(* IEC 61131-3 sources: ml2plc/benchmarks/st (part 24) *)

    bias_8 : ARRAY[0..63] OF REAL := [-0.00346507085, 0.0794098824, -0.0815823004, -0.0197601747, -0.0118380254, 0.0312293377, -0.00609452976, 0.00358696282, 0.00419461308, -0.0723088458, 0.0482314527, 0.0938620642, -0.0692073926, 0.0194631442, -0.0589119196, 0.0299020465, -0.00631620362, 0.00955793448, -0.0159860123, 0, -0.00618809368, 0.0138237355, 0.00124220713, -0.0202849712, -0.00431400631, -0.0275725052, 0.111446135, 0.11047177, 0, 0.0995986015, 0.0175163615, 0.0613925792, -0.00830586068, 0.00282396353, -0.0744342729, -0.0211106688, 0.0866850466, 0.0997213498, -0.00675268006, -0.0535650924, -0.0118874479, -0.0482638218, 0.00823871326, 0.0484990887, -0.0278981514, 0.0414009988, 0.0608626865, 0.0968099013, -0.0129826535, -0.0369008854, 0.00364142703, -0.0370340049, -0.00600347202, -0.0126274861, 0.0921183825, -0.0980235487, 0.00168389722, 0.0823842064, 0.0339883827, 0.0445966795, 0.0921582058, -0.0254019089, -0.0172969531, 0.0778813958];

    weights_11 : ARRAY[0..4095] OF REAL := [0.152399674, -0.263345957, -0.224488631, -0.188193366, -0.0617991723, 0.148717895, 0.0324863903, 0.114666007, -0.289823532, 0.0125278663, -0.0137963807, -0.022444414, 0.110561207, 0.119829476, 0.334477097, -0.139504924, -0.0269849207, 0.113053806, -0.0107069612, -0.180623204, 0.0457108654, -0.214532733, 0.0401020236, 0.00631321967, -0.167630613, -0.0481288582, 0.195484549, 0.111929268, -0.0581923984, 0.0258115064, 0.238763675, 0.0641915128, -0.0806587264, -0.224124625, -0.0460969172, 0.091414094, -0.013553381, -0.043530602, -0.0263040792, 0.140525028, -0.0622836426, 0.15601474, -0.497485936, 0.129424945, -0.170885473, -0.125799641, -0.339268953, 0.0710499883, -0.116152979, -0.0266817547, 0.126233891, 0.131714255, 0.290685475, 0.165184066, 0.283396602, -0.059989959, 0.0141595677, -0.136663362, 0.20351474, 0.0463219136, 0.00223265006, 0.0316324756, 0.182196692, 0.341547728, 0.0614045113, -0.00371772563, -0.275792897, -0.193623677, -0.0266438629, -0.103982933, 0.0405711122, -0.00346332369, 0.0464573167, 0.000740021234, -0.303002685, 0.0795986727, -0.0327266343, 0.0721366256, 0.147136018, -0.105440497, 0.101954572, 0.0728471428, -0.0363206528, -0.0158560108, -0.330246508, -0.212550044, -0.093112044, -0.197731018, -0.125574902, -0.078097105, 0.034774553, -0.262974173, 0.15699707, 0.14151752, -0.0313425213, -0.0470193997, 0.19462584, -0.255247116, 0.357496887, 0.000614301243, -0.195358515, 0.0303748176, -0.175757021, -0.0335321315, -0.0249454323, 0.0811241418, 0.0762640387, 0.116933405, -0.128208607, 0.00518320873, -0.029634852, 0.11359746, 0.017268436, -0.104347244, -0.115615718, 0.202678129, 0.10678266, 0.0986468866, 0.190590888, 0.0687514096, 0.0356852412, -0.0412406325, 0.0757317245, 0.0352434814, -0.342369705, -0.0480474308, 0.266226262, 0.0569148995, 0.0286941677, -0.2472938, 0.0204578005, 0.0296292026, -0.0654909462, -0.10515099, 0.151057318, -0.0363138504, 0.00139550562, 0.0611258186, 0.0148243103, 0.227309123, -0.0798782185, -0.11899174, -0.157541484, 0.314520597, 0.170248464, 0.265226632, 0.0593360811, -0.0398373678, 0.0081351446, -0.0901603773, 0.18755962, 0.00631602108, -0.207302138, 0.103253566, -0.240270436, -0.0895837396, -0.105462186, -0.135611624, -0.0793325603, -0.0249736756, -0.13815324, -0.0941773206, -0.189351335, -0.112737559, 0.293767184, 0.0163262729, -0.175204575, -0.0996527299, 0.231760427, -0.0418962091, -0.0648548007, 0.268336385, -0.032381732, 0.245270595, 0.0585076436, -0.0289969705, 0.232107788, 0.279983878, -0.011282769, -0.121292524, -0.295017779, -0.131171674, 0.0821883231, 0.216307148, -0.0106242169, 0.00658608973, -0.21936737, -0.139937028, 0.182932571, 0.233257622, -0.286341697, 0.246410012, -0.0386230387, 0.0858042613, -0.0830237195, -0.110467531, 0.0558926836, -0.0293775387, -0.216672435, 0.134263664, -0.0869384855, -0.0198220555, -0.0998319387, 0.122479506, 0.124716364, 0.12669073, -0.165978372, -0.0657829642, 0.0525778681, 0.0783382952, 0.0370095335, 0.141239166, 0.0418702848, 0.0749414936, 0.240086794, 0.0674306303, 0.0347193331, -0.0469557568, 0.041893255, 0.090664953, 0.0798208192, -0.124962248, -0.0150589822, 0.0606806017, -0.212737143, 0.0127978772, -0.0479948185, 0.193862215, 0.18940939, 0.110280916, 0.00163242826, -0.0205761306, -0.129006281, -0.141371146, 0.147304669, 0.0262788441, 0.167370602, -0.141203105, 0.200771987, -0.234238222, -0.149722278, 0.23931098, 0.0104937805, -0.266669959, -0.164157122, -0.041039072, -0.250695556, -0.112417288, 0.193107903, 0.140542001, 0.0903390646, -0.230039254, 0.0777369738, 0.260997742, 0.0930059701, 0.138459459, 0.0424353629, 0.171048418, 0.156789139, 0.0312985368, 0.133111879, -0.120839193, 0.0985307842, -0.175964057, 0.122762412, -0.117720641, -0.129174918, -0.104449466, -0.144933715, -0.215081707, 0.0680070445, -0.129005954, 0.0603452325, -0.0575148351, -0.203575164, -0.0453374311, 0.155170351, 0.106897905, 0.0749150291, -0.144247919, -0.171046615, -0.132302389, -0.147862911, 0.00684731873, -0.0410480648, 0.15876098, -0.190579101, 0.0498549677, 0.0963715315, 0.086084798, -0.0875354186, -0.153710201, 0.145764962, 0.0200527348, -0.100025706, -0.135493338, -0.0464859232, 0.00132688298, -0.0185684748, 0.0582565144, 0.187669724, -0.0816467628, -0.0872224793, 0.157934099, 0.0402881019, -0.0318563916, -0.142950997, -0.11230398, -0.0497585908, 0.161313683, -0.1942278, -0.0826544166, -0.0122894971, 0.0872979611, 0.0720221922, 0.0849900693, -0.177533969, -0.152409315, -0.100491337, -0.0112174684, 0.106480442, -0.0379864834, 0.0722993612, 0.163500831, 0.18924883, -0.135068297, 0.0942396447, 0.0284191072, -0.0632716715, -0.138580009, 0.193715364, -0.150715292, 0.0303814765, 0.111110657, 0.117106274, -0.0263905209, 0.0506038666, 0.0267103072, 0.0400604308, 0.154954746, 0.108434454, 0.0550541244, 0.0168840457, 0.0785695761, 0.0604145676, 0.144188315, -0.206482708, 0.0983125418, -0.0374258012, -0.00447623339, 0.205374479, -0.0380841345, 0.0740306601, -0.0350800455, 0.0866823494, -0.0981449634, 0.0656447932, 0.0974652469, 0.0593180098, -0.0401085094, -0.0922544375, 0.0644713044, -0.0637705103, 0.205211937, 0.27076602, 0.0604185574, 0.245794445, -0.0236300994, -0.027567558, 0.1355685, 0.0849664137, -0.138995841, 0.159796208, 0.0539290234, -0.0213833489, 0.0917554945, -0.193392858, 0.0205196254, -0.154481247, -0.0105813192, 0.158501342, 0.01522783, -0.0629718155, -0.222794086, -0.138768524, 0.00203081919, 0.170994595, -0.0148755405, 0.0800000504, 0.194157824, -0.113540575, 0.0917406157, 0.238140926, 0.00717910752, 0.21342735, 0.0675954148, -0.0781002492, 0.179200038, -0.0140909683, 0.217517018, -0.0182730798, 0.154534876, 0.130978897, -0.15910472, -0.242845848, 0.192364007, -0.0712619573, -0.172466293, 0.153321937, 0.196527407, -0.14488329, 0.0236006379, 0.0861952752, -0.0437985249, 0.175121501, -0.0954023749, -0.114573762, 0.143516839, 0.00525142904, 0.126135498, -0.116257451, 0.109212697, 0.0145286033, 0.104307882, -0.0975407884, -0.164253727, 0.0486553423, 0.0687329695, 0.187514946, -0.049572818, 0.0788708553, -0.0701822415, -0.045390375, 0.100607939, -0.0249090847, 0.0791288838, 0.154155806, 0.232392356, 0.110889055, 0.0298407078, -0.0190417878, -0.0341505446, -0.22469382, 0.0715206563, -0.109233215, 0.0421755537, 0.0418922678, -0.0328179933, -0.161357954, 0.0284879543, 0.0438218452, 0.257945627, 0.227448493, -0.129958495, -0.392283171, 0.109769329, -0.0173306819, 0.0859658271, 0.108519241, -0.0660175383, -0.0608303361, -0.0360111594, -0.0876427889, 0.190083712, 0.0288716163, 0.238107309, 0.136543661, -0.00705705583, -0.0259979162, -0.00647293031, 0.069024533, 0.0381969362, -0.152234167, 0.295585841, -0.401145488, -0.108133636, 0.209102049, 0.0307547674, 0.147690207, 0.128031835, -0.0473762713, -0.147987187, -0.164643124, -0.059981253, -0.14839074, -0.0456473343, -0.335970312, 0.0270624142, 0.273908377, 0.0461861901, -0.221928775, 0.151594713, 0.0270567555, 0.0552504733, 0.288964689, -0.075935334, 0.270585835, 0.235102609, 0.181183606, -0.116892524, 0.0349841826, -0.0259137452, -0.310423553, -0.0737684369, -0.224190742, 0.102769867, 0.148424283, -0.00051581359, 0.109018147, 0.131758898, -0.241935253, 0.0429472104, -0.192998812, -0.156563684, -0.199549347, -0.0259795301, 0.118114009, -0.202294961, 0.00430562347, -0.0795410797, -0.186826259, -0.12402641, -0.0973436236, 0.062623024, 0.0698438436, -0.0140991006, 0.0761193931, -0.157981157, 0.054249879, -0.0833289996, -0.119116187, -0.175815642, -0.193181172, -0.0350408033, 0.0374635346, -0.148473918, -0.111192934, -0.110237554, 0.0392782576, 0.0543338954, -0.212789983, 0.214189187, 0.261465758, 0.0389742181, -0.0119669382, -0.041862458, 0.0934221447, 0.154760599, 0.104591891, 0.135659441, 0.124115832, 0.125245571, -0.0981265381, -0.173501864, -0.225834534, -0.040620435, -0.0631992593, 0.11226812, -0.151412457, 0.0888080448, 0.130535215, 0.114341483, 0.0704539269, 0.238751054, -0.0625069663, 0.183925942, 0.162767082, -0.0624889433, 0.18303372, 0.0478743874, -0.214895129, 0.150446177, -0.0400604196, 0.164489478, 0.156864062, 0.280662, 0.0744856521, -0.109412298, 0.222006962, -0.188556612, 0.257241905, 0.00763767865, -0.0429345556, 0.000701996032, -0.256307662, -0.0537884794, 0.258199453, -0.145994559, 0.0452899151, 0.0317057781, -0.0876930654, 0.08571475, -0.092731908, 0.184803054, 0.18809928, 0.0703473389, -0.00392604945, 0.142104432, 0.160575241, -0.0699259192, 0.196616039, -0.160764754, -0.202707544, 0.150236309, -0.194807246, -0.142325938, -0.240276873, -0.0591731966, -0.0514629297, 0.00134343619, -0.166902661, -0.188654795, 0.0843883976, 0.0013771971, 0.169252023, -0.161208317, 0.208919898, -0.118219167, -0.24853687, 0.147254348, -0.040950682, -0.104150467, -0.182231963, -0.162871018, 0.0433620438, 0.126293465, -0.166178107, -0.186834484, -0.22719419, -0.216035366, -0.311863422, 0.10080345, -0.10563679, -0.21303615, 0.0257087015, 0.063385427, 0.0836621374, 0.137088358, 0.0247118175, 0.157823056, -0.162809089, 0.274433285, -0.0909785628, 0.219206274, -0.150779128, -0.206102833, 0.0196267851, 0.215949804, -0.080320105, 0.0171771869, -0.126778483, -0.169971392, -0.0758564174, 0.037309479, -0.184586704, -0.176283911, -0.0172518641, -0.223967373, 0.0620737523, -0.210962385, -0.0175580438, -0.198382184, -0.133766785, -0.192560017, 0.00918835402, -0.0767401755, 0.136367351, 0.171674535, 0.183295757, 0.220561728, -0.0821217224, 0.1140071, -0.127449334, -0.151443526, 0.118891813, 0.0171878282, -0.027197564, -0.0242941491, -0.232013106, -0.109213538, -0.117022179, 0.0856248662, -0.151049286, 0.142516539, 0.125007212, -0.156722993, 0.266981691, -0.130809814, -0.0616114177, -0.0442247763, 0.0877789408, 0.0459268093, 0.225089535, 0.059550181, -0.0352692939, -0.0199252516, -0.140248358, -0.181541502, -0.0301125441, 0.114853002, -0.155363366, 0.120270431, -0.119383417, 0.15385288, -0.137697816, 0.0990949422, 0.139819413, 0.101220191, 0.0159896575, -0.0617526323, -0.0679681972, 0.113188118, -0.042417895, 0.0258083455, -0.169725969, 0.075258702, -0.0537487082, -0.149268836, 0.109437704, -0.116023861, 0.0976026133, -0.215568498, -0.257916421, -0.0836541727, 0.0753511712, 0.194070086, 0.0318242721, 0.0160240829, 0.0868645757, -0.188116699, 0.181180835, -0.207172692, 0.110726506, 0.171905503, -0.121312834, 0.00326830451, -0.134259403, -0.244052947, 0.156338409, 0.239065826, 0.0572260544, 0.22199899, 0.0920382291, -0.0747542828, 0.0250579547, -0.209005356, 0.314894259, -0.0127276182, 0.188592002, -0.105892763, -0.203456968, 0.218186542, -0.0714133903, -0.090361774, -0.0645971596, 0.0143091576, 0.298341304, 0.159289271, 0.0570015721, -0.199153751, 0.019798452, -0.0419481322, -0.128920168, 0.0999377146, -0.245023876, -0.0517567694, 0.247462109, -0.070638895, -0.0811767727, -0.128980458, 0.11074882, 0.0168372188, 0.0593690798, 0.175101206, -0.054478053, 0.022643229, -0.307910532, -0.0983424112, 0.0169419218, -0.131076947, 0.295372337, -0.176049858, -0.0388735868, 0.261773378, 0.186196834, 0.0407921039, -0.060955897, 0.0722839534, 0.1541913, 0.118314162, 0.185275882, -0.0770900249, -0.186694846, 0.118786186, -0.022491321, -0.0364597216, 0.089644663, 0.0571428053, -0.253871858, -0.0122213988, 0.204711184, 0.312439799, -0.320880443, -0.27240929, 0.122102626, -0.273709536, -0.0164961014, 0.0607479513, 0.291678041, 0.223591253, -0.198138237, -0.118850462, -0.238560677, 0.323092818, 0.0589599535, -0.194248945, 0.00573190255, -0.0346102566, 0.00809514709, -0.1437345, -0.0768056959, -0.0114840511, 0.14923422, -0.0970238969, -0.0471924804, 0.0891452581, 0.176614508, -0.150917053, 0.31215173, -0.0488434397, 0.0310474988, 0.13556391, -0.210260242, 0.265471876, 0.127534941, 0.00403250754, 0.210733801, 0.0956179649, 0.0654093474, 0.0347067229, 0.0318550393, 0.248021692, 0.0198314767, -0.115047991, 0.108949013, -0.10042078, -0.29889968, 0.0146387629, -0.141234264, 0.204530731, -0.144104674, 0.105720773, -0.23340179, 0.0790494978, 0.18509376, -0.206608996, -0.0394043922, -0.0189410113, -0.230545685, -0.198211581, 0.220677823, -0.0647635758, -0.195251271, 0.201641157, -0.177163646, -0.095896475, 0.0920335501, -0.138604224, -0.109693781, 0.236355498, 0.0536849797, 0.115611076, 0.212027684, 0.0571522713, 0.240873307, -0.0458607674, 0.310614586, 0.233346224, 0.0570905395, 0.130410984, 0.169783399, 0.0727831423, -0.0302463956, -0.30536887, 0.0152019113, 0.163850963, -0.109125808, 0.0144169629, 0.132228628, -0.0707990453, 0.193070427, 0.165563926, 0.0941457525, -0.0627072603, 0.0423249342, -0.111638814, -0.0591745116, -0.0470574982, 0.29292962, 0.0765838027, -0.142371729, -0.112034045, -0.0560461804, 0.156755283, -0.235810399, -0.201336101, -0.125491038, 0.201229259, 0.123228803, -0.238689259, 0.0129049234, 0.0961765721, 0.0151871378, 0.266222477, 0.186487585, -0.217119902, -0.0869368389, 0.124067664, -0.065676488, 0.140951827, -0.198084503, -0.178457528, 0.0855591595, 0.1007246, -0.0287072621, 0.0854200944, -0.178427383, 0.0386579223, -0.0619194172, 0.09910997, -0.129233211, -0.068861261, 0.13413316, 0.139778435, 0.0833287686, 0.0622766875, 0.235616207, 0.201298133, -0.182556123, -0.00869753398, -0.047157418, 0.268308789, -0.225152835, 0.0152922235, 0.153030574, -0.0839851871, 0.167121798, -0.0833399519, 0.093423374, -0.0923105478, 0.178122193, -0.203960165, 0.0267385971, 0.0512525626, -0.22356531, 0.056387879, -0.0550887249, 0.161965206, -0.195818886, -0.0647771284, -0.182523564, 0.17741926, -0.116015404, -0.0489375815, -0.202825278, 0.147160143, 0.191247597, 0.0707065612, -0.00766302971, 0.170157924, 0.0735885873, -0.141567349, -0.21014148, -0.129353657, 0.0956847668, 0.0227197595, 0.0941244364, -0.0791912824, 0.107957929, 0.199303105, 0.0537132025, 0.0155240446, -0.147489786, 0.0846396238, -0.0715232193, 0.182592198, 0.00312403357, 0.0118206823, 0.0933757424, 0.162187204, -0.0768953189, 0.130623519, -0.154309347, -0.0370425209, 0.225373268, -0.0371935703, -0.512049019, 0.0894301012, 0.149142876, 0.0406918228, 0.054195568, -0.222945645, 0.125597313, -0.121843651, -0.192063659, 0.022529887, -0.129418507, 0.100320496, 0.14389959, 0.100439146, 0.211798623, -0.139967546, 0.104904346, -0.0939587057, 0.127366856, 0.138831839, 0.0239571333, -0.00880390406, -0.0611199997, -0.10359811, -0.0635057986, -0.00202414393, 0.188975051, 0.18646647, -0.133227944, 0.0697101131, -0.0743370131, 0.0876726359, 0.174912781, 0.132824585, 0.00545993866, -0.000499482965, 0.169128001, 0.219260916, 0.214551806, -0.0652708858, -0.0217023604, -0.193402603, 0.00403163396, -0.117414609, -0.0933148414, 0.00748919882, 0.200135365, -0.141633987, -0.214732349, -0.091433309, 0.204348087, -0.0532101393, 0.154062733, 0.248481318, -0.13802442, 0.192950904, 0.16888696, 0.149313912, -0.222851619, 0.153076321, 0.182242945, 0.185836926, 0.141479209, -0.0413135886, -0.0169824678, -0.0272292644, 0.089787066, -0.0702687651, 0.158348948, -0.0452950932, -0.0598885454, -0.174950615, 0.291644782, -0.0561419651, 0.0800843909, -0.215036035, 0.13363564, -0.103067927, -0.0768741667, -0.0631346405, 0.0626737475, 0.15906544, -0.327983201, -0.123729207, 0.19425182, -0.14580068, -0.110915102, -0.0493397824, 0.0671491474, 0.00072730938, 0.0883379132, 0.123690397, 0.189004809, 0.0893278271, -0.114139549, 0.308739871, 0.0107161012, 0.118270479, -0.337565839, 0.261260688, -0.0494029, -0.0752659142, 0.238311097, -0.108185798, -0.12475723, -0.0681707337, 0.0807750225, 0.0104115838, -0.0831196159, -0.161203995, 0.0769510195, -0.178012058, 0.165514678, -0.0196140297, -0.0373411514, -0.0155290961, -0.161595047, -0.0622068048, -0.291716814, 0.218920842, -0.128163859, 0.044695992, -0.187777534, -0.105463572, -0.0571242459, -0.0119509697, 0.00533423526, -0.0132009489, 0.161444128, 0.190533608, 0.136306271, 0.158209473, 0.215961605, -0.0804739892, 0.117368713, 0.126664549, 0.133364782, 0.152663857, 0.136497244, -0.336019129, 0.150216475, 0.20953989, -0.0419718549, 0.00763540342, 0.0507058874, 0.0899446309, -0.0746354163, 0.126670465, 0.0997138247, -0.131774053, 0.18959567, 0.186503679, 0.0671444461, 0.107626587, 0.125563666, -0.0331348479, -0.0831428245, -0.0118116708, 0.13317202, 0.179913059, -0.00435783528, -0.103403352, -0.169043481, 0.134726152, -0.143405557, -0.143480599, 0.145388424, 0.0501072556, -0.100935332, 0.0670109838, -0.0547590144, -0.11869137, -0.164782315, 0.14261204, 0.0516628996, -0.0139837861, 0.158076271, -0.0323812068, -0.0253638402, -0.0481653959, -0.166442499, 0.0914008841, -0.126121193, 0.10642685, 0.080969587, 0.195150837, -0.0635801703, 0.0927808583, 0.0660431832, -0.113444202, 0.2108161, 0.0454176217, 0.207712188, -0.158912182, -0.149667591, 0.225732028, -0.144124746, 0.220306486, 0.187320516, -0.056225121, 0.190556765, -0.184439331, -0.128877133, -0.0283655971, 0.148606017, -0.103650376, 0.0173259694, 0.0809403509, 0.00934745371, -0.129418105, -0.0100147277, 0.0515523404, 0.00264053047, -0.133236319, 0.213405624, 0.200618967, 0.011354222, 0.0573964044, 0.0985980853, 0.00135266967, -0.129998296, 0.151727006, 0.204372659, 0.200007543, 0.21404855, 0.189805731, 0.172358885, -0.0890808403, 0.0522677153, 0.107005432, 0.113238558, 0.0461152345, 0.119334862, 0.113662854, -0.202756092, 0.122567102, 0.156569704, 0.0166884214, -0.127153099, 0.130326495, -0.162898168, 0.0981043428, 0.199507132, -0.092357628, -0.0304451138, -0.156488106, 0.0427581519, -0.213457823, 0.157986298, 0.212126359, -0.191093981, -0.0687070787, -0.155501977, 0.075762704, 0.202147499, -0.0100540668, -0.0357479602, -0.165612519, 0.0348113328, 0.0888052136, 0.0522147566, 0.00634533167, -0.000127598643, 0.0748969465, 0.0386748761, 0.0424322337, 0.212277904, -0.0906898081, -0.0402118266, -0.14763388, -0.163068712, -0.00134003162, 0.0113786161, -0.114206046, 0.0614237338, -0.143889531, -0.096885711, 0.20141612, -0.20934172, 0.159835026, 0.0288719237, 0.0186812729, 0.0141171068, 0.202441737, -0.00636282563, -0.0913520604, -0.00343427062, -0.0776682198, 0.114591286, 0.178352684, 0.072447516, 0.207320198, -0.164817482, -0.133918926, 0.0607623905, 0.133606508, 0.108131513, -0.00368179381, -0.0975685716, -0.18251574, -0.12751992, 0.217671528, -0.00256840885, 0.0633859858, 0.0459913127, -0.0114317834, 0.019155506, -0.0564544499, -0.173174202, -0.0360071398, -0.161694646, -0.201523215, 0.143933117, -0.0519516505, -0.189812288, 0.0398772061, -0.0408333391, -0.180227458, 0.141621813, -0.115172304, -0.121136017, -0.0121303732, -0.204050809, -0.0434726924, -0.046715267, -0.0699533895, 0.171459943, -0.144236326, -0.0683937967, -0.0708762109, -0.102386728, -0.0776161775, -0.193716198, 0.186093926, 0.0237003118, 0.121066563, -0.125280246, 0.0977233648, -0.0399483182, -0.0141839087, 0.145612508, 0.0374964625, 0.0779918507, -0.0435630977, 0.0875028968, 0.071565561, -0.0101307984, 0.165002391, 0.201880664, 0.00914894603, 0.186509728, 0.170419008, -0.00774519145, 0.0486198589, -0.257243395, 0.0580342449, -0.123784639, 0.13865912, -0.172557667, 0.151741877, -0.101602815, 0.110366128, -0.120282121, 0.0840358585, -0.13807863, 0.135065734, 0.152518809, -0.213707358, 0.157859072, -0.0512838028, -0.119913951, -0.0603275895, -0.0344250649, 0.0280932616, -0.113776729, 0.00914250128, 0.169182256, -0.0726605803, -0.118695714, -0.162195101, 0.109512694, 0.214561909, 0.201593056, -0.0490923934, 0.231536657, 0.000906694273, -0.0773898289, 0.229626477, 0.292316675, 0.0434411876, 0.0439935587, -0.171945095, 0.168419257, 0.138824657, 0.187337905, -0.121906206, -0.121290758, 0.0895823315, -0.205835402, -0.102580823, -0.064769879, 0.0918552354, -0.0006545863, 0.0484051257, 0.00231042434, -0.1427017, -0.00512752309, -0.118499592, 0.167649359, 0.173335105, 0.0724587515, -0.0639462695, 0.189106256, -0.0253329333, -0.167535514, 0.199837193, 0.054232005, 0.173054591, 0.208212107, 0.063709937, 0.178403363, 0.102365844, -0.145370528, -0.0627328828, 0.204421952, -0.217216507, 0.152429745, 0.177940995, 0.123621874, 0.161663517, -0.0583134182, 0.113821968, 0.147727966, -0.0192146897, 0.120329253, -0.206288442, 0.118907943, 0.0558229275, -0.119626381, 0.115259588, -0.123966016, 0.189842731, 0.304001242, -0.133949921, -0.00190896366, 0.111900635, 0.194404766, 0.129541457, -0.0793663859, 0.0952215493, -0.205361709, 0.0308174528, 0.276944697, 0.150184885, 0.0571603253, -0.0862910375, -0.209261745, -0.00469737314, -0.107266292, -0.0262841173, -0.21763204, 0.0261462647, 0.0255539753, 0.159364834, 0.0638701171, -0.133363664, 0.166979283, -0.191513494, 0.167016715, -0.201660112, 0.0460934602, -0.00581953721, 0.00407372508, -0.078385748, 0.176348567, 0.261097163, 0.0668909401, 0.0932687446, 0.268428653, 0.111295953, -0.0538752489, -0.0353972577, -0.0643084422, 0.0826371983, 0.241673946, 0.0859841257, 0.0413935967, 0.192854241, -0.0863617063, 0.102388531, 0.0939005539, 0.110310666, 0.0338847861, -0.0237080809, 0.192427814, 0.00698334165, 0.0662905425, -0.134980679, -0.00617967499, 0.190878674, -0.00159786642, 0.0727328956, -0.240946233, 0.196102977, -0.0931468382, 0.0836528018, 0.103284612, -0.239004865, 0.0113834683, -0.129806876, 0.14836894, -0.232858315, 0.089459613, -0.179351673, 0.144995049, 0.196424425, -0.0279766843, 0.132153019, -0.105318397, 0.187499374, -0.00858527701, -0.0920507312, -0.11234127, -0.0994759649, 0.175084785, -0.0811289176, -0.100668162, -0.387158185, 0.153878331, -0.178559199, -0.119826905, -0.0257519037, 0.202533126, -0.165797308, 0.1972083, 0.0326090157, 0.191457987, 0.208948106, -0.0303138606, -0.168486714, -0.212763578, -0.00552030979, -0.0189667419, 0.196747944, 0.209965065, -0.14008227, -0.356117338, 0.0720864087, 0.2261962, 0.262177914, 0.190582126, 0.125341758, 0.131352305, -0.0850886703, 0.105056457, 0.0996146277, -0.364396185, -0.1066579, -0.145678446, 0.0647635385, 0.0825714245, -0.0452001728, 0.13121967, -0.145201892, 0.102415368, 0.160855427, -0.1157851, 0.176233247, -0.106195346, -0.17459546, 0.0715932772, 0.0647462085, -0.0499108769, 0.0551721789, 0.0756226256, -0.115369171, 0.115483992, 0.182759956, 0.134363547, 0.19813326, -0.00339539489, 0.22427693, 0.0874575227, -0.0538085252, 0.0250612367, 0.194358304, 0.0420459919, -0.197343454, 0.15234834, -0.0194482468, 0.207918748, -0.370312631, -0.191926241, -0.238808528, -0.0383893885, 0.126615122, -0.0540592968, -0.207585737, -0.0226110499, 0.0861546621, 0.258043557, 0.30580011, -0.265124172, -0.172527641, -0.0776732266, 0.0940554887, -0.0529039092, 0.22364676, -0.0504839607, -0.111994199, 0.0752739981, 0.167051509, 0.231486157, 0.222942859, -0.0696845353, -0.151163772, 0.250781924, -0.146447971, -0.0967529416, 0.184217557, -0.300973266, -0.126572028, 0.215180457, 0.187338904, 0.185731187, -0.11665196, 0.000876162725, -0.0202561766, 0.125354245, 0.10827215, -0.160607785, 0.188338622, 0.0980067775, 0.0324687324, -0.219831422, -0.168211251, 0.200699002, 0.1139713, -0.216335818, -0.0309214499, 0.0763551295, 0.0451243334, 0.0868523866, -0.000636569108, 0.0952483416, -0.11416243, -0.125886872, 0.0755488724, 0.107398666, -0.0849267319, 0.0167402681, -0.368645281, -0.106054433, -0.136857152, -0.113142923, -0.140909985, -0.0106369946, -0.0734956935, -0.242627531, -0.163561374, 0.0919052735, 0.125031963, -0.043657735, 0.0146407625, 0.153221101, 0.0668651685, -0.190944195, 0.0788392946, -0.0817975849, 0.124928646, -0.361474574, 0.110909373, -0.255627602, -0.142462447, 0.0353607163, -0.252555937, 0.194031313, -0.0276524629, -0.0741961077, 0.0262450166, -0.102495871, 0.107768953, 0.141406447, -0.322431296, 0.174083382, -0.174821675, -0.395054817, -0.0608991683, -0.341402888, -0.146280155, -0.290810555, -0.0700072646, 0.0340672284, 0.114190154, 0.212211475, -0.29652983, 0.0295428969, 0.194639176, -0.0198184811, 0.133799478, 0.138498858, -0.182915777, 0.0482293516, 0.0976990163, -0.18222487, 0.0835105181, -0.106537037, -0.0591551289, -0.115260668, -0.11497248, 0.0435057431, -0.159548879, -0.105683692, -0.260151893, 0.0550674088, -0.0321849883, -0.0744472593, 0.00243522367, -0.181820303, 0.252596408, 0.270988226, 0.168165222, 0.0595975779, 0.0989734977, 0.17273213, 0.0179654639, 0.013571118, 0.0022207133, -0.0643146485, 0.14008981, -0.0777452365, 0.134650469, -0.155961126, 0.0555896498, -0.0966854021, 0.0125770848, -0.000214683023, -0.151022673, 0.196903691, -0.115989923, 0.262134969, -0.0680010691, -0.224485368, -0.199625343, -0.210131735, -0.0643070862, 0.0685092211, -0.413198173, 0.0757171661, 0.0919734463, -0.359562606, -0.201385498, 0.0115947183, 0.174798757, -0.0814683214, 0.0596277267, -0.0625551641, 0.0350604355, 0.184136912, -0.164665803, 0.0183611717, 0.250624686, 0.0125863301, 0.0112502538, -0.0108454721, -0.0688611045, 0.16646485, 0.0284723155, -0.326143622, 0.251596063, 0.0676906854, -0.111148089, -0.0604397766, -0.357566506, 0.00267260056, 0.0472641513, 0.185109943, -0.0561866984, 0.148887575, 0.102317147, -0.0849794373, -0.0614579991, 0.0326576456, 0.0126584023, -0.0629983395, 0.223311111, -0.00327185332, -0.148226351, -0.183692589, 0.00595363649, 0.178311333, -0.14655976, -0.0530309901, -0.0653009266, 0.237797007, 0.173097223, 0.200525954, 0.131583318, -0.116117708, 0.0929283351, 0.098859176, -0.101166539, 0.211423203, 0.180236056, -0.098462984, 0.0356300026, -0.055087164, 0.070975855, 0.0152753443, 0.0117747337, 0.0124992579, 0.0186377019, -0.040137589, -0.174795151, -0.0888965726, 0.216044262, 0.173421398, -0.0901128203, 0.0402170271, -0.123981677, -0.0186401308, -0.120826356, 0.106725052, -0.19337979, -0.137401208, -0.123095892, 0.124976858, 0.151482031, -0.141049087, 0.0428393334, 0.174957797, -0.14806959, -0.0215549618, 0.186499581, -0.204556108, 0.210095719, 0.0789846629, 0.029979974, -0.108856134, -0.0139944702, 0.0263781548, -0.125280932, -0.10276451, 0.0262285024, 0.0617966205, 0.0358561426, -0.181433201, 0.116816476, -0.173377424, -0.181904286, -0.178747416, -0.00100579858, -0.141323447, -0.17858167, -0.215236828, -0.124892443, -0.18321009, 0.166554824, 0.0349302441, -0.0718755722, -0.21206364, 0.202988341, -0.262059748, -0.0846684426, -0.0264383312, -0.0190072507, 0.2202245, 0.128679246, -0.126438454, -0.0482899137, -0.136346161, 0.164990321, -0.0377886444, -0.00999837369, 0.145294696, -0.206945017, 0.168252572, -0.123122193, 0.0317248851, -0.0978919715, -0.111651219, 0.074932836, -0.281826913, 0.185020849, 0.055261448, 0.00178773759, 0.0390683152, -0.246171236, -0.0958288237, 0.210186899, 0.275020272, 0.0562327988, -0.133841649, -0.161592439, -0.0814305469, 0.151387647, -0.0924248621, 0.256124526, -0.0551051423, -0.211608618, -0.0358127393, -0.104693621, 0.1162875, 0.113921165, -0.0199713167, -0.23672004, 0.17288205, -0.0616145991, -0.167591259, 0.0158987548, -0.105777226, 0.00850734301, 0.206110939, 0.220944673, 0.173485622, -0.0885103047, -0.123291343, 0.119619459, -0.0967060253, 0.162609577, -0.23304899, 0.024063224, 0.0214320533, 0.2257936, -0.116359495, -0.0210717637, -0.0603798702, 0.0435092635, -0.00730895204, 0.103644289, -0.10791108, -0.00523050129, 0.0974855199, 0.250795186, -0.0883831903, 0.211329684, -0.0763134733, 0.0505424179, -0.194253653, 0.160468459, 0.0373329632, 0.00362053118, 0.232644767, 0.0308330338, 0.161484063, -0.0271853432, -0.131138071, 0.11403884, -0.0388104171, 0.0234489087, -0.0291281473, -0.16315636, 0.238832727, -0.125655994, -0.051028531, -0.150253788, -0.0957489237, 0.161308855, -0.010553672, 0.145903602, 0.178950518, 0.206775278, -0.197363213, 0.100926705, 0.127155304, 0.0886795744, 0.0384771898, -0.0636024028, 0.136744395, -0.0296712294, 0.255500585, 0.0886330456, -0.015306036, 0.127241626, 0.0978040919, 0.00628852937, 0.0744743049, 0.213523507, -0.0189819261, -0.104008943, 0.028438326, -0.0549609102, 0.108124904, 0.0547557399, -0.0689821094, 0.282766223, -0.0776696652, -0.145231634, -0.219961882, -0.0325948037, 0.170671925, 0.238952041, -0.220119491, -0.0539352782, -0.205213696, -0.0961958393, 0.0955754817, 0.190853387, -0.106655076, -0.0676123053, 0.207522944, 0.0059924447, -0.136339933, 0.170324996, -0.0170212891, -0.186595798, -0.122996755, 0.0536680296, -0.124922357, 0.0955476314, 0.0518711582, 0.176927432, -0.112219326, 0.100288011, -0.117357753, 0.199554503, 0.0488559753, -0.0699957237, 0.228910819, 0.00692145294, -0.0817696825, -0.108787522, -0.128030986, 0.0173476879, -0.131096452, 0.236910611, 0.0257094558, 0.255908877, -0.018263232, -0.00103016174, -0.0486674346, 0.073059462, 0.244683802, 0.0431794897, 0.0152821513, 0.168885887, 0.108368844, 0.167778686, -0.213540077, -0.211735442, 0.105609275, -0.0604555644, -0.155116454, -0.196209759, -0.0379836187, -0.0647224784, 0.00641336106, -0.14297466, -0.107331365, 0.183396488, 0.184337839, -0.0531041622, 0.00186734158, 0.244511604, 0.0740732402, -0.0291328561, -0.0445070565, 0.144737765, 0.0123820817, 0.11382781, 0.197113797, 0.201976836, 0.245440185, 0.119564258, -0.146405488, 0.117127948, 0.0338072814, 0.190734386, -0.25059697, 0.199911967, 0.207614452, 0.0533561595, -0.0374337807, 0.142019153, 0.0490953773, -0.216328979, -0.10855855, 0.115646183, -0.263035089, -0.148798853, 0.124370195, -0.13782458, 0.124930479, -0.116868503, -0.0248529781, 0.0512323603, -0.0528448075, 0.0193750132, 0.192962959, -0.152398363, -0.0119206896, -0.0373266339, 0.0179096516, -0.0443546325, -0.0742346868, -0.0461954102, 0.294702619, 0.154465228, 0.0773186088, -0.310861647, -0.0707053468, 0.266035378, -0.0992082134, -0.332212776, -0.205583721, -0.196842909, -0.281396747, 0.136664137, 0.201202393, -0.139625281, -0.0458463132, 0.186710879, -0.129951373, 0.130285919, -0.235751554, -0.0895666406, 0.199424937, 0.0833966285, 0.135916606, -0.108947381, 0.00343655213, -0.116784215, -0.189424649, 0.235676333, 0.225083172, -0.0404505059, 0.0241782386, 0.138108522, 0.141151369, -0.180884242, -0.070838213, 0.0613366216, -0.134111598, 0.025904512, 0.201248944, -0.128643408, 0.12299782, -0.132246569, 0.249260843, -0.18512398, 0.17548199, -0.11300002, -0.368429303, -0.0116485134, -0.0219518971, -0.187667757, -0.0626360103, -0.028858915, 0.153726026, -0.104429685, -0.266087621, -0.209274143, -0.186508, 0.180915117, 0.156441614, 0.203999043, 0.144177482, 0.10513787, 0.0303519256, 0.133759394, 0.192577541, -0.140958086, 0.237446681, -0.237315372, 0.0912553743, 0.172334418, -0.11051251, -0.380104393, -0.185993105, -0.231100082, -0.0684015378, -0.165600955, 0.194090798, 0.0481378883, -0.139796764, 0.130825281, 0.172460839, 0.265127957, -0.112289988, -0.0345997512, -0.167480007, 0.0347576514, -0.0154025862, 0.0508864224, 0.138450637, -0.143623456, -0.216727793, 0.0870179385, 0.152233243, -0.218138441, 0.134071931, -0.105602548, 0.0766346306, -0.210313886, 0.173437417, -0.0167097338, 0.176717728, 0.260095805, 0.0725469142, -0.0281031746, -0.0118673686, -0.23178342, 0.196914256, 0.207952037, 0.0597638041, -0.0669040531, -0.202766195, 0.105974823, -0.196885899, -0.130043596, 0.0408547632, 0.051734861, 0.150090992, 0.126557499, 0.0610106736, 0.0459405072, 0.217397436, -0.178916857, -0.235516325, 0.257763088, 0.0747808293, 0.144583955, -0.205134392, 0.245919466, -0.208999187, 0.260882437, 0.132566705, 0.150488973, -0.00251174299, 0.13973631, 0.0961362347, 0.177716032, -0.0470190607, -0.0734431297, 0.0359828062, -0.00525023043, 0.102971934, 0.0987021625, -0.173347533, -0.00715078134, 0.127415687, -0.0373299271, -0.204287812, 0.178136423, 0.138002157, 0.0237582866, 0.174087659, 0.240981013, -0.116837405, 0.130510405, -0.000766741985, -0.124521762, 0.261766434, 0.236482263, 0.087483488, 0.248471096, -0.0924688652, -0.0650356933, -0.0104683442, -0.0764830336, -0.209237933, 0.0235566385, 0.124604762, 0.106890164, 0.159328818, -0.0968483388, 0.100116894, 0.12527816, -0.213597402, 0.0560539104, -0.121492833, 0.0191260874, 0.126306266, 0.0674194768, 0.0697287023, 0.0672566965, 0.0521879978, 0.053629946, 0.205602214, 0.0651868656, -0.0143089797, 0.175055593, -0.143693537, 0.184233233, 0.245637834, -0.0019021834, 0.0554781668, 0.122372709, -0.0944118276, -0.00765591115, 0.246960357, -0.0359783396, 0.013843908, 0.250939488, -0.0550113358, -0.0771496817, -0.129822791, -0.0721774176, -0.287194103, -0.0553002506, -0.0833646432, -0.0302243531, -0.209284484, 0.0714682192, 0.174552351, -0.00634080404, -0.255132675, 0.0539513268, -0.171819359, -0.130697995, 0.0328636803, -0.172556356, -0.2824184, -0.0451180376, 0.0577123426, -0.192122251, 0.0324847363, 0.00184812211, -0.140389964, 0.0564051718, 0.0673946068, -0.0826997831, -0.218807384, -0.226912007, -0.0740968361, -0.0628938675, 0.0246492196, 0.0681713596, -0.344983399, 0.0526000336, -0.31024906, -0.206341609, -0.216349587, 0.0267339684, 0.122782297, -0.178241864, -0.0923086107, 0.0223308429, 0.136397615, 0.248619109, 0.200533465, -0.293138444, 0.311404914, 0.239410847, 0.0427243561, 0.252901375, -0.0671737939, 0.0358522087, -0.101214036, -0.0909479931, 0.312909693, -0.0543796271, 0.225179315, -0.30917415, -0.0924400315, 0.233333379, 0.0843650997, -0.160150632, 0.179808214, -0.0429063886, -0.0673761442, 0.215058282, 0.171212927, -0.0550884008, 0.142365858, -0.110932022, -0.169926539, -0.0976140499, -0.0154480785, 0.0212051291, -0.0351677053, 0.020173341, 0.0828600079, 0.0684699938, -0.140169322, 0.12288864, -0.249438584, 0.161289573, 0.183076456, 0.0643565208, -0.0405365787, -0.003901063, -0.0275522638, -0.114001192, -0.344557256, -0.0885162503, -0.06081542, -0.332393795, 0.277116388, -0.0268625468, -0.190394998, 0.21460636, -0.215998247, -0.222107425, -0.255408615, -0.136359274, -0.14687404, 0.142695963, -0.140400141, -0.0201289766, 0.0542479455, -0.00637657382, 0.137159288, 0.123378307, 0.173221618, 0.0176266842, 0.0871137902, 0.314738423, -0.24674274, 0.139450938, -0.0980865434, 0.0819776729, -0.202197522, 0.0445437841, 0.0490690246, -0.248550311, -0.235274941, -0.334431201, -0.0380337983, -0.0726476014, -0.166573018, -0.0421880521, -0.231450424, 0.130716771, -0.0721551031, 0.11855723, -0.14029862, -0.0331737548, -0.018478848, -0.0687058344, -0.1540602, -0.107552357, -0.146992445, -0.246584743, 0.264962852, 0.0624919087, -0.0870190263, 0.115786649, -0.114350855, 0.212790087, -0.20117563, -0.0133681539, 0.204012766, 0.191788897, -0.0210248157, 0.115564667, 0.113092259, 0.174278691, -0.148719802, 0.190654084, 0.0438634008, -0.0724180192, 0.134725466, -0.123058394, 0.162449196, 0.204366207, 0.116563216, -0.19426021, -0.0909457207, 0.199671999, -0.118528321, 0.117968924, 0.109732315, -0.0419445187, 0.00864718016, -0.0645976812, 0.0311101824, -0.109628826, 0.111323684, 0.014768647, 0.208999589, -0.094222419, -0.179808035, -0.0267504808, 0.109660603, 0.217561051, 0.106540732, -0.00727470964, 0.0496581346, 0.134096339, 0.0660558417, 0.167213649, -0.0612058528, -0.0911486596, -0.0100888135, -0.155831024, 0.189135149, 0.156071231, -0.00602033734, 0.0703240484, 0.0744462162, 0.0984698087, 0.140996054, 0.124672696, -0.163873687, 0.0303707868, -0.199095607, -0.0432972983, 0.0943269432, 0.0672637746, -0.0916577727, 0.0945999026, 0.271431386, -0.146770418, 0.228228882, -0.088630408, -0.221145526, 0.201267377, -0.0209989715, -0.205188558, 0.0660831109, 0.165487453, -0.110452496, 0.0229095519, -0.023997318, -0.0244352669, 0.0483070128, 0.0403944179, 0.00371245272, -0.026503861, 0.00920362957, 0.130575255, 0.185562894, -0.150229856, 0.208181933, 0.066503644, -0.14963977, 0.183380142, -0.0742605925, 0.0525272898, -0.207853332, -0.150708884, 0.0244787, 0.118969277, -0.244963139, 0.108839378, 0.370168149, 0.162852734, 0.0989103541, -0.13296926, 0.045421198, 0.0944304913, 0.0636059344, 0.0407316796, -0.128235891, 0.211519986, 0.188827261, 0.0511491187, 0.00440762937, -0.0511926375, 0.0151363136, -0.112162314, -0.0530756265, -0.261404067, -0.0806499943, -0.114475191, 0.092728734, -0.112707078, -0.186766997, 0.16012606, 0.137830883, 0.170057893, 0.185820624, -0.140461251, -0.213634878, 0.125510231, -0.215242818, 0.0796449333, 0.132684961, -0.2006073, 0.0357116349, 0.198004097, -0.0991434678, 0.0635548085, -0.215833962, -0.0722895563, -0.108518705, -0.051846981, -0.137091249, 0.120727405, -0.0786514506, -0.0299482532, -0.0290962607, -0.0490365773, 0.156231463, -0.0395558923, 0.0900194496, 0.128394648, -0.0630546808, -0.0585276112, -0.205579251, 0.160481736, 0.0202968903, -0.163621709, -0.0748255625, -0.184875816, 0.125386044, -0.127115071, -0.143687502, 0.091046527, 0.0920635611, -0.0941656902, -0.173573211, -0.0986982659, 0.0191576183, 0.0842896551, -0.209140688, -0.0771613792, 0.168761611, 0.0210189521, 0.129767984, -0.0285845138, -0.202819064, -0.209608585, 0.0455416664, 0.167025864, 0.163965836, -0.132653818, 0.0619048737, -0.0682924837, 0.166164339, -0.127146959, 0.166915938, -0.199976191, 0.0883914679, 0.122442588, 0.157862335, -0.0999033526, 0.107905447, 0.271243006, -0.0405978113, 0.181895465, 0.10665185, -0.0172348171, -0.263982832, -0.0332699679, 0.253317565, 0.263973176, 0.151911378, 0.0881777182, 0.22092396, 0.1231746, -0.152555913, 0.101217501, -0.179812282, -0.047235027, 0.064411968, -0.100622997, 0.134386688, -0.197145775, -0.0489049777, 0.00595416129, -0.0711699873, 0.0988756642, -0.25260219, -0.135066882, 0.178719059, 0.0527570769, -0.217263788, 0.0104796821, 0.141307697, 0.192717046, 0.0233423207, 0.0181158278, -0.0247748066, -0.1053892, 0.0186107531, 0.0304267742, 0.247790694, 0.0885608569, -0.165538073, -0.0982961208, 0.078451246, 0.0747933313, 0.149838224, -0.294142485, 0.204276547, 0.0315016098, 0.148058638, -0.0792296454, -0.00655980362, -0.0633319467, -0.134122044, -0.0603130311, -0.228715405, -0.0372798219, -0.0637207702, -0.00131563691, 0.0267799813, 0.205451921, 0.0369303524, -0.194896266, -0.146388203, 0.0251822565, 0.10831248, -0.304889441, -0.067542769, -0.0279039573, 0.224844977, -0.0980764031, -0.177602947, -0.11175137, -0.233728245, -0.223739907, 0.0452572368, 0.0688700527, 0.0517109595, 0.0646637455, 0.0814413205, 0.185665578, 0.199086443, -0.045935303, -0.206678033, -0.110741898, -0.0746753067, 0.0203328282, -0.0121729225, -0.32386151, 0.317199111, -0.000200206137, -0.0206671208, -0.0143212825, 0.109568812, 0.127662241, 0.148976833, 0.134836257, -0.0659915805, 0.0971495807, 0.129318729, -0.261195183, 0.139618188, 0.175515547, 0.177529424, -0.0397923216, -0.171056911, -0.152844191, -0.256262839, 0.0387250036, -0.109484434, 0.348202139, 0.181829244, -0.0921679214, -0.14175418, 0.351582646, 0.0428714491, 0.109188475, 0.113643356, 0.190801248, 0.0840984732, 0.0745595545, 0.202311695, 0.110946044, 0.0192239713, -0.138841808, 0.142307326, 0.354664713, -0.0450815856, -0.107993297, -0.03863943, -0.0024780829, 0.0134169487, -0.117628835, 0.0603437982, 0.166732147, -0.118978985, -0.163896814, -0.0940616056, 0.139851525, 0.0401148871, -0.000361859042, -0.0329533368, 0.00609338423, 0.0956700072, 0.0159509256, -0.183647871, -0.0647861436, -0.0180492532, 0.126684785, 0.174701124, 0.00719110668, -0.0489515066, 0.151985407, 0.0191572756, 0.103651136, 0.0472620092, 0.0433273539, -0.0642805994, -0.117137074, -0.117250271, -0.217558905, 0.238560513, 0.156538591, -0.201861724, 0.252844602, -0.153291538, 0.0394916683, 0.131754085, -0.168700293, 0.282408744, 0.0575271547, 0.270327926, -0.210436061, 0.136073276, 0.0850231051, -0.187773168, 0.179164112, 0.0486085825, 0.131480142, -0.0669804588, -0.12845093, 0.136758476, 0.183792964, -0.0880155787, -0.0198557992, 0.0737654716, -0.150122464, -0.181854174, -0.0218842644, 0.244106069, -0.0331436694, -0.118402436, 0.112792633, 0.161135405, 0.193292305, 0.0654401034, 0.151135877, -0.105567589, 0.163530335, 0.0537123606, 0.115299411, -0.107796557, 0.144485876, 0.190182522, -0.225720987, -0.188096419, 0.0644563586, -0.219243228, 0.0506861359, 0.0646403879, -0.155654714, 0.0720595792, -0.0648836493, 0.0587573051, 0.115380988, -0.144375831, 0.193385601, -0.216615528, 0.0823164284, 0.121625237, 0.0662951022, -0.104674295, -0.0913950354, -0.0744329914, 0.0588016734, -0.0569245294, -0.123344973, -0.112728342, 0.0536800511, -0.0440075137, 0.00869007315, 0.231819123, 0.180460185, 0.112645507, -0.151289985, 0.170129269, -0.118003756, 0.0397904888, -0.0155688487, 0.000529384532, 0.16991967, -0.0197017621, 0.0159432869, -0.152901173, -0.141727105, -0.209757477, 0.0510494262, -0.206472322, -0.125095367, -0.144546479, -0.213549063, -0.0514436178, -0.0335596912, 0.141235679, -0.224663511, -0.0350644737, 0.0376378372, 0.17774488, 0.188020244, 0.0334532149, 0.155813828, 0.0600071736, -0.0559457168, -0.0678997114, 0.0960994884, -0.202544078, -0.157427654, 0.0421013534, 0.115875132, 0.152794838, -0.12245059, -0.152902767, -0.212830245, -0.124761559, -0.202095598, -0.0178206097, 0.126928881, -0.0542535968, 0.128561482, 0.212066635, -0.144553557, 0.0753035396, -0.1383304, 0.0503492504, 0.265743077, 0.227717698, 0.131189972, 0.0942342579, -0.0386557281, 0.00459791953, -0.151728719, -0.0490803644, 0.170358211, 0.107892729, 0.027722558, -0.0222314857, 0.0439844616, 0.0846926421, -0.136754051, -0.126678228, 0.0100780185, -0.00410804106, -0.0236090273, -0.235840544, 0.116327874, 0.12390665, 0.154099762, -0.0710356757, 0.0358319879, -0.00236812909, -0.056195125, 0.0473820642, 0.121515736, -0.12424425, -0.177752599, -0.165439278, 0.0420489013, 0.13842456, -0.122449316, 5.4429478e-05, 0.0483980328, -0.198470056, -0.0108445771, -0.129893675, -0.102530636, -0.0193273257, -0.14624238, 0.08766298, 0.0668683425, -0.133514196, 0.0853877515, -0.0655543208, 0.133385897, 0.00266161677, -0.10532745, -0.0290171318, -0.00419039, -0.00792111829, 0.0604869053, 0.00910193752, -0.118941627, -0.12992464, -0.172481984, -0.012415126, 0.165430143, 0.0105601074, -0.0124265226, -0.204574227, 0.0933492258, -0.0265834965, 0.0440250263, -0.120509379, -0.237719804, 0.141081452, 0.251164675, -0.00922667235, 0.0145384986, -0.23117803, 0.120755881, -0.0217975043, 0.120932087, 0.0436988175, 0.000108511711, -0.174057677, -0.0660731643, -0.0309707671, -0.133766994, 0.115545824, 0.188281238, 0.153618366, 0.0869733766, 0.126192153, 0.0268286113, -0.138225377, -0.106887072, -0.0767892227, -0.220131189, -0.119694576, 0.00380183011, -0.226367459, -0.111844957, 0.152785808, 0.242726147, 0.106298521, -0.248363763, -0.32967785, 0.105129965, -0.155959815, 0.138976559, -0.00137228239, 0.0948434696, -0.0816367492, 0.0710474625, -0.418901235, 0.135055959, -0.310039103, -0.0387624092, 0.249349698, -0.416977942, 0.0891338736, 0.00944569428, -0.237012804, 0.0804961771, -0.195645198, 0.0945587382, -0.0762844086, 0.0416320711, 0.00949457288, -0.127774417, 0.259676754, -0.40856576, 0.0794008449, 0.0908604041, 0.133119613, -0.100699835, -0.156859353, -0.162409276, 0.00788537692, -0.0637622774, -0.32110858, -0.134144261, -0.206960112, 0.0118728764, 0.0764703378, -0.394238651, 0.183452353, 0.241670236, -0.141249031, -0.16704978, 0.018816743, -0.0430508442, -0.170661062, 0.176272959, 0.16203025, 0.23600857, 0.149680734, 0.0821367577, 0.175770909, -0.126697093, -0.148051918, 0.190101504, -0.0317378193, 0.0456583053, -0.270201981, -0.0483634844, 0.319031864, 0.0222948454, 0.0767141506, -0.00711641507, -0.153200984, -0.143897697, 0.140922055, -0.0283886902, -0.113231972, 0.139692098, 0.142846361, -0.157825753, -0.100115009, -0.0507604778, 0.0704903975, -0.0313803554, 0.161187619, 0.0637935027, 0.154604718, -0.178512841, -0.108615682, -0.119129255, -0.0183542315, -0.200408816, -0.06402006, 0.0961765796, -0.183909222, 0.103326656, 0.12906833, 0.175179169, 0.075670667, 0.138392508, -0.121290363, -0.0992279351, -0.141292989, -0.0473258048, 0.130663127, -0.147083119, -0.123233199, 0.203898117, -0.204678267, 0.167588547, 0.158947214, -0.115444884, 0.0865047872, -0.162406579, 0.00433421135, 0.0109670609, 0.0494914539, -0.0845709294, -0.0436661392, -0.0943619311, -0.133204848, -0.133604929, -0.0241765436, 0.0312332567, 0.0160661489, -0.192561835, 0.170536771, 0.0699443966, 0.18987824, -0.198280796, 0.13675791, -0.128286049, 0.133142799, 0.0423047841, 0.19421573, -0.0902426615, 0.045400776, -0.0236111488, -0.0612643398, -0.0522969365, -0.185536757, -0.0624252073, 0.0719867498, -0.145684376, 0.342741668, -0.169891864, 0.189545587, -0.20563516, -0.106448837, -0.00803494453, -0.139683664, 0.239471704, 0.347251058, 0.0986964926, 0.191767052, 0.0345206708, 0.117405772, -0.0646648407, -0.0939145163, 0.0358834863, -0.14516075, 0.329907864, -0.245812029, -0.20081225, -0.128157064, -0.32458353, -0.202067211, 0.310102135, -0.259800404, -0.183582872, 0.348934501, -0.00135924411, -0.00762309879, 0.0397878811, 0.0435562618, 0.190664694, -0.219969705, 0.167273611, -0.0363034643, 0.0843212157, -0.0630743131, -0.127757251, 0.133702457, 0.241022587, -0.0452217422, 0.157935485, 0.0468397252, -0.184891075, 0.0217796862, -0.174830914, 0.0529149808, 0.0344027728, 0.0301657226, -0.0991806537, 0.0966322273, -0.0987405106, 0.0616976731, 0.037891306, 0.144457489, 0.293943793, 0.125130758, 0.279702634, 0.2190516, -0.0891123265, -0.319427043, 0.020325454, 0.198740065, 0.244544879, 0.150971532, 0.139485016, 0.155953914, 0.100290887, 0.039516408, -0.11156898, -0.239001468, 0.0233942177, -0.0897894874, -0.0399748348, 0.141847938, 0.0783665776, 0.00495733274, 0.020279035, 0.166984901, 0.280435681, -0.217270985, 0.185803846, 0.191354558, 0.0111610517, 0.1644153, 0.0352947488, 0.0664995685, -0.0161591228, 0.0244116578, 0.0823068097, 0.0366923697, 0.20036611, 0.0597134568, 0.0136301629, 0.0214036219, 0.0707080811, -0.0257597454, 0.141371503, -0.0871877447, -0.0384720117, 0.159895733, -0.271953613, 0.118647724, -0.0838832259, 0.14117156, -0.0238901209, 0.0837025568, -0.0994942114, -0.311766535, -0.0361485183, -0.173598096, -0.0820912719, -0.109803088, -0.202099934, 0.13466467, 0.298355758, 0.147975996, -0.0162965041, 0.0887476951, 0.0656182021, 0.158688262, 0.00327817141, 0.216407076, 0.0288510714, 0.0746814311, 0.0788815916, 0.183364213, 0.149168417, -0.0533465818, 0.120975912, -0.0698309764, -0.131480917, 0.0775775313, 0.190101609, -0.175806463, 0.208605766, -0.0509476848, 0.0475929938, 0.172246516, 0.128037199, 0.135146201, 0.04195638, -0.179263756, 0.191762373, 0.124527775, 0.18047376, 0.0364429019, 0.133441925, -0.0794005841, 0.152522027, 0.0759226233, -0.194360182, -0.11856693, 0.0628863648, -0.140197754, -0.118163697, 0.148727104, 0.109244518, 0.0861630365, -0.0484799929, 0.144106314, 0.0300433505, 0.159115046, -0.0456953831, 0.159014627, -0.230968624, -0.191417232, 0.079684414, -0.0845753998, -0.216385618, 0.1015696, 0.12075875, -0.195914701, 0.0704701394, 0.00612893514, -0.172618523, 0.14040117, -0.0350932516, 0.0685307756, -0.0815743059, 0.0343151689, -0.226708308, 0.0161583424, 0.00600387063, -0.0403283834, -0.200709447, -0.136831269, -0.0756262839, -0.0913945809, -0.00991040468, 0.0491666384, 0.181557953, -0.0815197825, -0.1748669, -0.105041094, -0.024442181, -0.137364954, 0.213511899, 0.114984736, 0.141203478, 0.191028729, 0.209437281, -0.117445506, -0.211069152, 0.213400275, -0.00855989754, 0.0147007108, -0.17848292, -0.160719216, -0.169281244, -0.00666991761, -0.12999402, -0.017418623, 0.0077680028, -0.096811451, 0.0399670899, -0.099848032, 0.00562751293, 0.0391903967, 0.144329935, -0.0322996452, 0.142276108, -0.0690825805, -0.215008646, 0.0819310695, -0.147535652, 0.157100156, -0.100781769, -0.191613704, -0.178416789, -0.164667308, 0.029264966, -0.00163395703, -0.157853901, -0.0132551193, 0.0478072613, -0.149802342, 0.168672904, 0.0820260644, -0.120356776, 0.0662041232, -0.183392614, -0.178459927, -0.156899661, -0.164349243, 0.209907949, -0.115875721, 0.0444762632, -0.201963484, -0.0449665599, 0.198717207, 0.198328122, 0.0849034563, -0.103813514, 0.117308304, 0.0936804041, 0.0462679416, 0.0836406723, -0.0418322682, 0.0411524326, -0.190647915, 0.0886535197, 0.211842492, -0.0770319477, -0.0116216559, 0.147017792, -0.0120076491, 0.0194121003, 0.138708234, -0.120179571, -0.0352452397, -0.028329812, 0.0094909966, -0.00187779963, -0.0943269953, -0.078908205, -0.0844167471, -0.197576553, 0.121277407, 0.210520267, 0.141214922, 0.0709877908, 0.185094103, 0.119538829, -0.0926069394, -0.0566524863, 0.17638126, -0.0237376336, -0.135814071, -0.136954382, 0.119367145, -0.203730926, 0.00643029623, 0.167091712, 0.179837942, -0.10910327, -0.0022002249, -0.169260845, -0.0575643629, 0.0475613885, 0.114217445, 0.0275517702, -0.15122728, 0.000335678458, -0.201629221, -0.191943482, 0.0599358231, 0.215006664, 0.157104149, 0.123682573, 0.199631587, -0.193868354, -0.253842771, -0.192569867, -0.450649053, -0.13617, -0.0669108927, 0.111150347, -0.00369961141, -0.191271275, -0.237755463, 0.181265593, -0.132041126, 0.157904267, -0.0143442852, -0.395011663, 0.0413822122, -0.119375452, -0.274717003, 0.0961166471, -0.392918706, 0.138946593, -0.406194896, -0.126115769, 0.103300825, -0.0749610662, 0.187398925, -0.0632039681, -0.0863866061, 0.222676188, 0.219102636, 0.28613168, -0.187663198, -0.416728288, 0.0453014523, 0.244026601, -0.129714295, 0.295904279, 0.085724242, 0.0173482616, 0.17430979, -0.268255919, 0.0690714642, 0.0642987117, 0.0120566841, -0.298500836, -0.250954837, 0.0702187121, -0.439573526, -0.121676624, 0.167861462, 0.185528114, 0.26526314, 0.27663222, 0.25443691, 0.0214734077, 0.161424711, 0.144671425, 0.157419518, 0.182189599, -0.0776689202, -0.0120218601, 0.271168381, 0.156823754, -0.127337053, 0.0545059741, 0.128410771, -0.148533046, 0.0630049855, 0.0160781369, 0.151448995, 0.101595782, 0.0654489025, -0.167899147, 0.13213931, 0.0983135328, 0.0369849391, -0.194617927, 0.0153781129, 0.270563185, 0.0342637785, 0.0746257529, 0.211298779, 0.154260978, -0.119062982, -0.0627138913, 0.259788841, 0.117369875, -0.0632641613, -0.137389138, -0.2181786, 0.174714953, -0.0711210594, -0.237840936, -0.0302677024, 0.0867897719, 0.185713023, 0.240260184, -0.186787859, 0.0108405575, 0.0771833137, -0.141014621, 0.147447675, 0.252978861, 0.0547764972, -0.0874451548, -0.31400758, 0.118284583, -0.199673429, 0.111848548, -0.214292303, -0.0464315489, 0.230785057, 0.18862094, 0.0352876596, 0.00474979123, 0.0109337727, -0.0291237906, 0.122409284, 0.128479972, -0.105726346, 0.106454507, 0.1788349, -0.0558397211, -0.0373482071, -0.0495012775, 0.0530157499, -0.163363129, 0.202189162, 0.0545998327, 0.157361299, 0.214383185, 0.107534043, -0.200028911, -0.125518799, 0.216706932, 0.230916902, 0.250411302, 0.146487787, -0.01959024, -0.140795499, -0.0633696094, 0.0885654092, 0.0913219228, 0.0871412084, -0.0358804837, 0.0180488303, -0.0806887895, -0.0637854189, -0.190897569, 0.136343226, 0.0202956051, -0.0698644817, 0.239365906, -0.306738168, 0.180551901, -0.0763572007, 0.0489863828, 0.00122147053, -0.0715313926, -0.173467308, -0.174637392, 0.170282349, 0.186628222, -0.00949032791, 0.00133445614, 0.011871323, 0.00409735739, 0.0181704815, 0.117498547, -0.129429266, 0.120077997, 0.216407701, 0.180566475, 0.232433349, -0.0555412471, 0.189128026, -0.151290759, 0.180261225, -0.321341038, -0.101906769, -0.174282476, -0.286496341, -0.0306703895, -0.115755208, 0.171560839, 0.127792448, -0.0103189619, -0.0854421407, 0.20230858, -0.135044008, 0.137085229, -0.0906790271, 0.206210405, -0.109169461, 0.221058965, -0.203725383, -0.223818555, 0.00837364979, 0.0698773786, -0.11478246, 0.0962926373, -0.0567478091, 0.194004565, -0.0646269023, -0.230514511, 0.121396624, 0.051594045, 0.0810926184, 0.11312753, 0.117401369, 0.0351090729, -0.101227865, -0.0286359861, -0.152758554, 0.195657834, -0.129182458, 0.255799025, 0.0658524111, -0.133879721, 0.135263368, -0.117422193, 0.259024024, 0.12137039, 0.0429658368, 0.161656618, -0.109413959, 0.0212555416, 0.00380118797, 0.0245974474, 0.0452777967, -0.109418437, 0.0556083173, -0.0991568714, 0.240161121, 0.131009638, 0.21446988, 0.0535303056, 0.0080528371, 0.0592104085, -0.117336079, 0.101440094, -0.180672362, 0.153361961, -0.148895979, 0.123094238, -0.20419763, -0.00546182692, 0.169995323, -0.0374472365, -0.0513039343, -0.100886956, -0.144634396, 0.226476029, -0.123933963, 0.082715638, -0.0514412038, -0.137042806, -0.0798420236, 0.295484096, 0.14945595, 0.0148293832, -0.141559213, 0.152552426, 0.110004902, 0.264642984, -0.182816103, 0.203673571, 0.0767816678, -0.0460664965, -0.0965382606, 0.00824740529, 0.00633397093, -0.0335266478, -0.00525524374, 0.0221320633, -0.144528076, -0.181572482, 0.186975211, -0.0915289372, 0.0789494962, 0.0443420336, 0.0566833429, 0.0106719388, -0.153921574, 0.0117017636, 0.0780537501, 0.172404632, -0.0487603694, -0.0259934999, -0.112953916, 0.013087403, 0.199101657, 0.0694961324, 0.099969998, -0.0189182963, 0.137308478, -0.00687692454, 0.130568698, 0.157788232, 0.0861073285, 0.195408612, 0.237710238, -0.0510148071, -0.127946258, 0.0196243692, 0.0884056464, -0.229083344, -0.0584382601, -0.0112535618, -0.056976635, 0.207119659, 0.0605573431, 0.170117199, -0.0873071477, 0.0375184156, 0.0693956614, -0.0853421167, 0.168883324, -0.246331498, -0.15294233, -0.0786210001, -0.0727810487, 0.230497375, -0.124767907, -0.0180434044, 0.152893081, -0.176393285, -0.135040537, 0.012329434, -0.066455029, 0.0633047223, -0.168565243, -0.169502109, -0.223331943, -0.168321326, -0.0599934012, -0.0564355031, 0.199666232, -0.193147793, -0.0922575146, -0.0880292282, -0.181692928, -0.200924233, -0.170735195, 0.138240859, -0.0760595798, -0.0921700075, -0.166161865, -0.0384436809, 0.0141204651, 0.130763844, 0.105647944, 0.153559715, 0.212668225, 0.0108604385, -0.019111041, -0.140727684, 0.150457844, 0.1883111, 0.221798778, 0.112573713, -0.165191919, 0.0167138427, 0.24837476, 0.165022895, 0.240100026, -0.0641816482, 0.156478882, 0.19513236, -0.0954566598, 0.0913641751, 0.0593185239, -0.123686202, 0.053503748, 0.0152200609, -0.153226435, -0.145596594, -0.0840086117, -0.179127425, 0.0691409111, -0.0299637914, 0.152311578, 0.0949365795, 0.00141828961, 0.201368794, -0.174666852, -0.0636612177, -0.171069294, -0.13758266, -0.182560191, -0.137745142, -0.127387106, 0.148039132, -0.000196392211, 0.176657051, -0.127840057, -0.0359740965, -0.0467125587, 0.00534770545, -0.0455735289, -0.177512407, -0.173216969, 0.162237197, 0.04842823, -0.178101718, -0.0483464934, -0.167974755, 0.0910376757, 0.184863344, 0.174440339, -0.133150682, -0.120608732, 0.217321798, 0.269066572, -0.138795853, -0.0962826163, 0.141585678, 0.243578151, 0.226173848, -0.0334078334, 0.0868586823, -0.236201584, 0.0429105237, -0.00714816013, -0.183364853, 0.0685243681, 0.0485652611, 0.211708516, -0.145325571, -0.0299601406, 0.0740182772, -0.17283687, -0.146753222, 0.0394501612, -0.102561951, 0.279482722, 0.234896556, 0.136510789, -0.0687329471, -0.146247506, 0.166320026, 0.088236481, 0.0455387309, 0.0368321836, 0.0928156599, 0.251261562, -0.202283695, -0.0876553059, 0.188739464, -0.1219403, 0.0595511906, -0.0864975601, -0.0519133434, -0.159869671, 0.255505502, -0.0236511845, -0.099469468, 0.146673471, 0.00879366975, 0.202414125, 0.200698897, 0.118802421, -0.0520094372, -0.194901958, -0.0494996794, -0.132057235, 0.0713604391, 0.166914493, -0.103728242, 0.173196629, -0.108285852, 0.130671516, 0.00665229931, -0.216195241, 0.00278148265, 0.150077969, 0.0377425104, -0.109352857, -0.0078518251, -0.143112957, 0.237058267, -0.24492383, -0.232783735, 0.0026126157, 0.0566774793, -0.217854828, 0.158665374, -0.141393185, 0.240377933, -0.0147471335, 0.105589516, -0.132414341, 0.269156039, -0.0360066108, -0.279901594, -0.070857726, -0.000133716909, 0.0994284675, -0.399730533, 0.0423182473, -0.0807459578, -0.364677131, -0.173550189, -0.201698035, -0.150411874, -0.104539521, 0.0632497221, 0.0475217737, 0.106961772, -0.0748255625, 0.0537245125, 0.150076792, 0.100195438, 0.160947844, 0.136155531, 0.0336693786, 0.00195461512, 0.0391892754, 0.155441701, 0.0603906885, -0.0828605369, -0.188219786, 0.01371055, -0.108915485, -0.188475981, -0.00214913161, 0.209178224, -0.0138332155, 0.106863379, 0.17023693, -0.104419991, -0.0188917425, 0.124385007, -0.112276614, -0.0786361247, -0.047841236, -0.249989852, 0.157759428, 0.0704554766, 0.0761716887, 0.124297529, 0.132825673, -0.0735627264, 0.202956781, -0.0342735052, 0.110366948, -0.150816396, 0.152661726, -0.146618992, 0.171531007, 0.0614210069, 0.077137284, 0.0930158645, -0.143225402, -0.158822253, -0.251074195, 0.135286197, -0.0735299885, 0.244000822, 0.113809302, 0.116750523, 0.051723171, 0.183311462, -0.137916028, 0.0244293083, -0.088045761, 0.0404897481, -0.0778224021, 0.131730989, -0.0429636389, 0.115714654, 0.0684564859, -0.044515267, 0.00754295383, -0.050703045, -0.129571319, -0.187777609, -0.16493459, -0.126211151, -0.0829479098, 0.0330205783, 0.243688241, 0.13541998, 0.0975747928, -0.206415966, -0.0957572684, -0.0585407391, -0.195936382, 0.123246349, 0.13101624, -0.196200132, 0.0490147881, -0.0278630313, -0.224047154, -0.20703429, -0.0990627408, -0.115552947, -0.419253439, 0.0287015885, -0.0131201446, 0.16262652, 0.122940429, -0.308744431, 0.117334351, -0.00441871164, 0.158816338, 0.171548396, 0.0269443281, -0.146471247, -0.013632034, 0.217089698, -0.228731453, 0.0371344909, -0.157528311, -0.0783996806, 0.00250388891, -0.308794379, 0.221041724, 0.121599473, -0.219423294, -0.411408722, 0.115201004, -0.142029077, -0.111949541, -0.151291326, -0.0684362724, 0.147531658, 0.108987704, 0.28183502, 0.207470536, -0.0262030065, -0.0661180243, -0.0931391194, -0.0792838484, -0.211057425, -0.32554251, -0.183445573, 0.00182158989, 0.121516146];
    bias_11 : ARRAY[0..63] OF REAL := [-0.00635589194, 0.0714284107, -0.0793445706, -0.0154935429, -0.0884047896, -0.00860749092, 0.015439475, -0.0443723239, 0.0648666918, 0.0137735978, -0.0558123514, -0.0234004352, -0.0720951036, -0.0323092379, -0.0251345523, -0.0864192247, 0.0349380858, -0.0508749001, -0.101302393, -0.00825020857, -0.0878332034, -0.0217018481, -0.0879978016, 0, 0, -0.0321543552, 0.0255989321, -0.0501851514, 0.0153964404, 0.0969368443, 0.0876909047, 0.0749777704, -0.00993307587, -0.0840824917, 0.107733645, 0.0926610008, 0.000463146862, 0.0615399294, -0.0173791237, -0.00302339089, -0.00108950492, -0.0433365181, 0.0978755206, -0.0621731691, 0.0341274589, -0.0879570246, 0.00440526195, 0.00455495017, -0.0902555734, -0.0262572207, -0.0154181952, 0.0162822157, 0.0986388773, 0.0995882377, 0.0237515792, 0, -0.0163629819, -0.02235475, -0.00682879193, -0.0143427243, -0.0962111577, 0.0128893042, 0.0858025402, -0.00971365813];

    weights_12 : ARRAY[0..4095] OF REAL := [0.106257081, 0.00435368251, -0.200017139, -0.170659184, 0.140568718, -0.121934257, 0.121075258, -0.16430898, 0.0690469891, 0.0433366559, -0.062450733, -0.20864369, 0.149895057, -0.0887060761, -0.0112437466, -0.137328371, -0.182793975, 0.00182112318, -0.192540094, -0.0729949772, 0.0874842256, -0.199801773, 0.161684632, -0.20927608, 0.18800509, 0.0292491615, 0.1377161, -0.00336401165, -0.0864470974, 0.13110055, -0.151119724, 0.182269529, 0.177959964, 0.145959258, -0.153364599, 0.208557755, 0.107231423, -0.122332707, -0.0526105985, -0.0178942829, 0.171287671, 0.0380937643, 0.210034788, 0.114255026, -0.176481709, 0.159083605, -0.0201071408, -0.0995351151, 0.158686295, -0.121905096, 0.0662830025, 0.145770177, -0.202360839, 0.108805642, -0.00403741794, 0.0131892227, -0.110621646, -0.0315053463, 0.0544626564, 0.0432279147, -0.0527887791, 0.0743454844, 0.000725448132, 0.13499485, 0.249794126, 0.201496869, -0.105599739, 0.115793243, -0.0131411431, 0.0381885171, 0.0861910731, -0.127799913, -0.0971342772, -0.12288598, 0.262936473, -0.178271964, 0.0656890273, 0.0264430493, -0.112000212, -0.0541253053, 0.0306299999, 0.030385958, 0.188352376, 0.216451868, 0.0554085672, 0.0997735932, -0.0144361956, 0.293800294, -0.2299909, -0.0211171489, 0.0223787352, 0.207233086, 0.164753318, 0.177156463, -0.0375560075, -0.0163145456, -0.0929765627, -0.104105949, -0.0902710557, 0.251464099, 0.178618342, -0.289695442, 0.0912541896, 0.120610818, -0.046938058, -0.0419063605, -0.189616457, 0.0257992372, -0.130752474, 0.205490381, -0.194339946, -0.151713759, -0.17453213, 0.178030372, 0.173221558, -0.0263473187, 0.186066285, -0.153767124, -0.00557854539, -0.177357957, 0.270246536, 0.203962401, 0.238550261, -0.148142517, 0.269313812, -0.0103741148, -0.183588952, -0.193594933, 0.162554562, -0.115353428, 0.0583416782, 0.0762180537, -0.09497796, -0.214766502, 0.139911622, 0.131524205, 0.00997098256, -0.11585062, 0.164202839, -0.320977002, -0.0759125501, -0.0785337314, 0.0255053025, 0.128980473, 0.0306141712, -0.126000479, 0.107428253, -0.118020132, 0.138766393, -0.284001321, 0.170607731, 0.102398202, 0.148915827, 0.160759792, 0.110466659, -0.252095222, 0.139449462, -0.315892965, -0.244656861, -0.123431899, 0.170097247, 0.321350873, 0.175645128, -0.206368536, 0.175698891, 0.00147240586, 0.29501459, 0.0298838075, 0.296299219, 0.187590197, 0.212566584, 0.11760661, 0.0084051853, -0.10937953, 0.149446264, 0.106912412, 0.118477888, -0.116064332, -0.0906607434, 0.0801626742, -0.060745582, 0.118430406, 0.241397575, -0.199510291, 0.1551781, -0.296400189, -0.0104944538, -0.145789325, -0.129684851, 0.0872599632, 0.0820529014, -0.00545078563, 0.218558997, -0.143248811, 0.192341313, -0.201770559, 0.0760860071, 0.106566764, -0.0349904001, -0.00749497209, -0.162278533, 0.247534171, 0.103120431, 0.123288512, 0.166345581, -0.0299496409, -0.244585529, -0.0239745378, -0.0884519145, 0.00908797327, -0.186777309, -0.0307503436, 0.0863535553, -0.029496571, 0.132126838, 0.0579786561, -0.00642398978, -0.0869056135, -0.130231008, -0.0773765892, 0.241189286, -0.0329741426, 0.00026981649, 0.196063191, -0.00166879594, 0.163482696, 0.0171640627, 0.214319944, -0.199893922, -0.0535125323, 0.118300594, -0.342376232, 0.12815164, -0.0961666852, -0.210583001, -0.26564607, 0.176150426, 0.109022953, -0.0346871875, 0.0834982768, -0.189139843, 0.0655928552, 0.091176711, 0.260871142, 0.140941069, -0.0211790819, 0.18120195, 0.180467978, 0.24436079, 0.15343453, 0.288015127, -0.0526540764, 0.196438268, -0.090705663, -0.138662577, -0.251701206, 0.137427241, -0.215658352, 0.0927336663, -0.161177158, 0.185746282, -0.143332213, -0.125291377, 0.217623547, -0.229488418, 0.0239045564, -0.12882176, -0.117315933, 0.127802238, 0.0137906745, -0.092000097, -0.113476872, 0.0914460868, -0.00983959343, 0.0662833154, -0.250207067, -0.0580342449, -0.122949809, -0.00861869287, -0.0351496413, -0.138369471, -0.120193399, -0.181908339, 0.1659161, 0.161926165, -0.243621573, 0.0815375894, -0.22421664, -0.200593099, 0.0567479655, 0.0271451306, -0.143274829, -0.200878218, -0.131388023, 0.264421344, 0.0492096022, 0.0876826793, 0.214776635, 0.0356173888, 0.108095407, 0.0600323044, -0.00878227595, 0.0185248479, 0.167779326, -0.167263448, 0.133649796, 0.0860351771, -0.0738951042, 0.167534858, 0.182380617, 0.0853289813, 0.126694575, 0.0129384911, 0.169833899, -0.119239196, 0.163785785, -0.0672808215, 0.15020664, 0.0820419118, 0.170347661, 0.100519873, 0.100219205, 0.0340493061, -0.20067209, -0.136349007, -0.114618428, -0.19835715, 0.0851126164, -0.147766441, 0.162698075, 0.192914501, 0.188429147, 0.0658050552, 0.034532465, -0.0661727563, 0.13281174, -0.0711044297, 0.0274692085, -0.19102478, 0.106214181, 0.193854347, 0.0253953449, -0.0946320966, -0.166038856, -0.0701704547, -0.203632638, 0.0977531224, 0.0993859842, -0.162032917, 0.0353222936, -0.0693225861, -0.213332132, -0.0769920498, -0.0619540252, -0.170087278, -0.0315041505, -0.0012934655, 0.152092174, -0.164900064, 0.0507530719, 0.152842164, -0.120405428, 0.077816084, 0.11334984, -0.129420042, -0.0410492569, 0.141592532, -0.118363351, 0.135873318, 0.104652397, 0.103805363, 0.20919849, -0.213056386, -0.123535939, -0.0476374961, -0.12322703, -0.0815903842, 0.043837294, -0.104243912, -0.019641865, 0.19847779, -0.0767066404, 0.0687408, -0.18236804, -0.0714362264, 0.0506636314, -0.110496551, -0.0978325754, 0.072953321, 0.00686401874, 0.0755573437, -0.123891488, 0.315234214, -0.154309481, -0.241670758, -0.320736408, -0.0229317304, 0.100737318, 0.0693938807, 0.00485423952, -0.212198153, -0.269200683, 0.111313589, -0.147343546, -0.0591220744, -0.314041585, -0.104359977, -0.196067065, -0.199609593, -0.062965855, 0.282515615, -0.0779074356, -0.0812170208, 0.237137318, -0.167712182, -0.0139279505, -0.229874283, 0.134501129, 0.0717539415, -0.0137814144, -0.207121581, 0.245981425, -0.163413405, 0.223312944, -0.112920046, 0.10596218, 0.128136829, 0.223039329, -0.0331489667, -0.155040503, 0.181968331, 0.0779197216, -0.0980575457, -0.179500878, -0.145538241, 0.112551749, 0.0494974405, -0.0378191695, -0.06296812, 0.135410845, -0.231428131, 0.027612973, -0.211544007, -0.222097173, -0.198571667, -0.042331215, 0.00269386172, 0.173073843, -0.106698252, 0.108658753, 0.231999084, -0.0199163556, 0.0840402842, -0.164054617, -0.169759646, 0.23305276, -0.097792089, 0.0453311168, 0.0280471761, 0.128820732, -0.119299456, 0.115963653, -0.0075415466, -0.112931721, 0.0670242161, 0.302933872, 0.017848229, -0.0486157276, -0.0201860815, -0.0808905512, -0.0494740121, 0.19418247, -0.223715872, 0.204738364, -0.268613338, -0.0106582586, -0.118218318, -0.109672047, -0.0247898009, -0.152243793, 0.117515177, 0.237196997, -0.170047969, -0.143073574, 0.0319675468, -0.291564047, 0.0861566067, -0.139199525, -0.128801718, 0.255365193, 0.143989652, -0.308390856, 0.00239204685, -0.0202191174, 0.121472307, -0.170474201, -0.174699128, -0.165195644, 0.310387254, -0.0541064925, 0.190462306, -0.0273283124, 0.122453421, -0.0220364239, -0.0813105553, 0.197180018, 0.104430646, -0.150599644, 0.307831496, -0.1770574, -0.1636246, 0.0556599572, 0.262393951, -0.182958364, -0.118844286, -0.163353726, -0.0945671052, 0.11168465, 0.0820354596, 0.0180940349, -0.135421559, 0.185812682, 0.258482575, 0.132772148, -0.0373393223, 0.0624215081, 0.0671000555, -0.261657447, -0.130482182, 0.132579386, -0.190884918, 0.041321177, -0.197137892, 0.0326368958, 0.256414056, 0.0671977028, 0.0115289818, 0.0246465355, -0.0270507559, -0.182449952, -0.0699588656, -0.153745219, -0.16926384, 0.0633526966, 0.0229592621, 0.164385095, -0.111254871, 0.0148687335, -0.0871399641, -0.30644083, 0.0704381168, -0.302938342, 0.163136542, -0.163225174, 0.161171958, -0.241714865, -0.0642526448, 0.153364688, 0.102497257, 0.14832598, -0.117911123, -0.22630614, 0.182896242, -0.0571457483, 0.146639496, -0.0514917709, -0.141151905, -0.192691699, 0.0471394546, 0.0913215056, -0.152800024, 0.0426181071, -0.0565117002, 0.00609446457, -0.193988711, -0.0499040708, 0.0436979197, 0.0999253839, -0.0795054361, -0.103425018, -0.209491357, 0.197339267, 0.11044497, 0.204888374, -0.320532471, -0.126293123, 0.151542276, -0.174009621, 0.0993844345, -0.000349115813, -0.281020701, 0.00936588086, 0.0860493854, 0.220661372, 0.170487523, 0.238573328, 0.0244113728, -0.0152693167, 0.200015113, 0.0352645107, -0.237889886, -0.116291612, -0.0838106349, -0.0905120596, 0.218899921, -0.127314493, 0.0822635666, 0.138225093, 0.0179952085, -0.15195632, 0.124049164, 0.092439875, -0.1056609, -0.0491449945, -0.0414935164, -0.141843528, -0.0563498996, -0.0736364797, 0.0624214932, -0.0850778669, 0.17593126, -0.0441847481, -0.155779913, -0.0650813878, 0.0375658721, 0.133375734, 0.0923169106, -0.0893951133, 0.0897832513, 0.0213206448, 0.239664406, -0.148517206, -0.030231189, -0.0527165271, 0.22417976, 0.169856504, 0.296273053, -0.212572232, -0.20888643, -0.016295081, 0.101754785, -0.0549197085, 0.211681917, 0.218397483, 0.18634066, 0.126820177, 0.0505925268, -0.0614112951, 0.0752623454, -0.10380286, 0.0540275797, -0.204340652, 0.145865679, -0.0346987806, 0.065127641, 0.0127901398, 0.199785799, 0.177719668, -0.183774799, 0.0209528748, 0.103368029, 0.0971299931, -0.127705738, -0.212714925, -0.0891776234, 0.15857552, -0.190184981, 0.00605630968, 0.0196366478, -0.153378323, -0.0976148546, 0.0536283739, 0.178155646, -0.0522708073, 0.243760437, -0.256778598, 0.159023032, -0.0108456258, 0.0449721664, 0.00447948091, 0.155550942, 0.0962128639, 0.0743119419, -0.123430736, 0.212962896, 0.0239776131, 0.0913750753, -0.13022694, 0.214200482, -0.0275251269, -0.0230850372, 0.0584084429, -0.137045443, -0.149423778, 0.293362677, -0.231559619, -0.155231133, -0.0807164013, -0.0462920144, -0.117076352, -0.108108059, -0.204536229, -0.0108255595, -0.013456245, 0.264667422, 0.0911884233, -0.181063846, 0.191370711, -0.0283466205, -0.1479083, -0.164247975, 0.191607475, -0.103012457, 0.110606916, -0.000815605745, 0.158466443, 0.00851375796, -0.0969890356, 0.126110435, 0.155427545, 0.189703301, 0.0150730461, -0.182569697, 0.241557285, -0.0367574021, 0.17438066, -0.0277641099, 0.151728004, -0.208000898, -0.134433463, 0.107581556, 0.0131943412, 0.128248185, 0.139681146, 0.026148105, 0.241393596, -0.106327146, 0.0285313632, -0.00392851001, 0.26787442, -0.0786702111, -0.0199960638, 0.0751241669, -0.177954569, 0.179708481, 0.260549545, 0.161560953, 0.0470447503, 0.120685622, 0.140657887, -0.123638831, 0.194805682, -0.0563831925, -0.209175766, 0.0824169368, 0.0606862344, -0.171402454, 0.193776771, -0.00800510868, -0.0670984313, 0.0924971923, -0.101887502, -0.0226375572, 0.240748838, -0.0621666946, 0.0973561406, 0.04852999, 0.183064163, 0.26137805, -0.259445339, -0.0423310697, 0.238807201, -0.159126639, -0.260159343, 0.0155518148, 0.139621124, -0.185930684, -0.167278677, 0.153316975, -0.0289743431, -0.0626375005, 0.120228775, -0.138989061, -0.15610528, -0.122687519, -0.145005405, -0.122514747, 0.0639393106, 0.118220925, -0.0740523934, 0.304092497, 0.0344584249, -0.123333976, -0.0309291482, -0.156307325, -0.0993042886, 0.122875266, -0.0432663597, -0.168591157, -0.281338513, -0.043137081, -0.117354706, 0.134987041, -0.14579919, 0.0790656805, 0.0152693419, 0.286864221, -0.135996044, -0.00733812153, 0.0475724824, 0.292973101, 0.00887088105, 0.112235606, 0.157097444, 0.224297404, 0.0614821911, -0.20666416, -0.00968252309, -0.184044868, 0.114056982, 0.0753099993, 0.0102361599, 0.244052678, -0.207539141, 0.0548489466, -0.167633072, -0.0237612631, -0.231893212, -0.0243409649, 0.164452314, 0.0128334379, 0.0672746599, -0.118385501, 0.0196032487, 0.00372122228, -0.0901152939, 0.0240558926, 0.0934285447, -0.0222456753, -0.185950816, -0.170683146, 0.072074756, -0.0274260845, 0.0501453765, 0.0197149329, -0.166320279, 0.123482324, 0.123843014, -0.109266885, -0.013747978, -0.00779475272, 0.155238539, -0.182944626, -0.0116707738, -0.00189979863, -0.0371467322, 0.000649258494, -0.0684414059, -0.0617489815, -0.0876107141, -0.171610132, 0.113506228, -0.188258782, -0.0664495453, 0.0116472142, 0.115066245, 0.213201389, -0.188051775, 0.157321677, -0.17768763, 0.117324159, -0.163545921, 0.210153237, 0.166902661, 0.0325763598, 0.208137721, -0.00108235527, 0.174134597, -0.0782251731, 0.148419902, -0.0446081758, 0.062131986, -0.0802285075, -0.0112878159, 0.191592947, 0.154550329, -0.130775481, -0.0966541022, -0.0837484226, 0.198908642, -0.100747377, -0.00711986143, -0.105124243, -0.116811574, 0.00965594593, 0.01702323, -0.0357450061, 0.217188969, 0.241389364, 0.112407587, 0.156611636, 0.155096814, -0.192019671, 0.244446054, 0.195701391, 0.22498773, 0.226725683, -0.0261454489, 0.0961467847, -0.160606489, 0.142043069, -0.0130630685, 0.0523964949, -0.0840317458, -0.149799123, 0.100000717, -0.198448598, -0.169559553, -0.146289423, -0.0743390396, -0.0182770509, -0.201591939, -0.0772255585, 0.104011148, 0.153238833, 0.190954477, -0.107943065, 0.0712087154, 0.0700664073, 0.113094702, 0.199309185, -0.158572003, -0.0452618487, 0.223115429, -0.11665412, 0.200311944, 0.272724211, 0.21544452, 0.18986252, 0.0543463267, -0.0146445958, -0.0732405484, 0.0544527434, -0.071323432, 0.0412523821, 0.15092124, -0.044222407, 0.0139736934, -0.206451863, -0.169845477, -0.117359452, 0.0564284809, -0.107622862, 0.056094747, 0.0175767932, 0.0678091124, 0.205945954, -0.199567676, -0.131202608, 0.116727181, 0.00307112304, -0.0610344894, 0.304451853, 0.246360987, 0.00679735234, -0.0727391765, 0.105304509, 0.0813725963, -0.0503737293, -0.0423749015, -0.0600213148, -0.0395135209, 0.242647633, -0.0567225255, -0.0953626633, -0.000300093001, 0.0312304609, 0.173153102, 0.0520930588, -0.304377019, 0.0964622498, -0.0814322978, -0.0572857037, -0.124899499, 0.173855051, -0.126501203, -0.0713063776, -0.0373672135, 0.150735512, -0.237116978, -0.139013276, -0.218322858, 0.0921640545, -0.0520263836, 0.257865846, -0.151795939, -0.120246775, -0.108947575, 0.280953765, -0.112184592, -0.0690225884, 0.128942892, -0.00621310109, 0.150983855, 0.265627414, -0.0148573527, -0.00638692081, -0.270087361, 0.0936407074, 0.119968422, -0.168551922, 0.065900743, 0.163260669, -0.0762269944, 0.121191658, -0.227582991, 0.0563046262, -0.14453648, -0.247026324, -0.198427394, 0.146938384, 0.0399760678, -0.00455863774, -0.00801403075, -0.00471097231, 0.129436374, -0.00785559881, -0.23967573, 0.160759911, -0.217170179, 0.059673205, 0.0550655685, -0.0963633731, 0.0493823029, 0.0798566714, 0.109029189, 0.020367872, 0.135246068, -0.113844417, 0.00287559745, -0.209072962, -0.197916552, -0.180231661, 0.101901092, 0.214207754, -0.00789650623, -0.106650531, -0.126928777, -0.0627369136, 0.0654484034, -0.0819197819, 0.29193005, -0.0248275623, -0.0557257682, -0.00748233451, 0.180867657, -0.0344851837, -0.250930518, -0.104754284, 0.147129387, -0.188409835, 0.169326276, -0.160357788, 0.169476837, 0.0106401676, -0.0722912773, 0.22912693, 0.229926616, -0.278435051, -0.00473464234, 0.0555630922, 0.17146723, -0.117122836, -0.0767989457, 0.0572060272, 0.142129436, 0.00657555461, -0.0285110623, -0.260344118, 0.0989044905, -0.105224997, -0.225994274, -0.282512605, -0.132227853, -0.23164551, -0.126432598, -0.175983578, 0.207563102, 0.20213519, 0.116067044, -0.129871324, -0.0641780123, -0.197573081, 0.0170770157, 0.0416710302, 0.237090498, 0.0815810338, 0.199073792, 0.0989497602, 0.170951322, 0.192848817, 0.02512151, 0.0494165868, -0.0813700259, 0.143076003, 0.136122361, 0.175064206, -0.161730811, 0.182675511, 0.0577683002, 0.12183997, 0.0470225997, -0.231185332, 0.0169506967, -0.119522803, 0.0683735013, 0.0920851454, -0.217990443, 0.0190431885, 0.203925014, -0.207395673, -0.0615044907, 0.0312225744, -0.073792249, -0.229524866, 0.155897632, -0.162459046, 0.0172525812, 0.136289224, -0.111660883, 0.237077177, -0.178375512, 0.175627097, -0.0281897094, 0.0541172661, -0.109059267, -0.14404507, -0.124059416, 0.0811684206, -0.0470161177, -0.066804871, -0.0850931481, 0.0434931368, 0.1373014, 0.259490013, -0.0881389454, -0.0493104868, -0.19704245, 0.16196382, -0.13053143, -0.111271337, -0.0854118466, 0.224985242, 0.127444759, 0.0727540329, -0.0320677198, -0.0183699485, 0.00351795973, 0.164765865, 0.13210772, 0.049928043, 0.0186676942, 0.0988922641, -0.131334722, 0.177617058, -0.170443878, 0.0973633751, 0.00504548103, -0.0171984043, 0.187171161, 0.0827463046, -0.157445848, -0.204074711, -0.245190218, 0.245169774, -0.0603508018, 0.17393136, -0.0305710733, 0.0401617177, 0.147684678, -0.0304231029, -0.152545437, 0.0501171015, -0.233973876, 0.136166081, 0.188226268, 0.0445944853, 0.0289832689, -0.202041328, -0.174103916, 0.131884769, -0.201908588, 0.221570641, -0.0861945599, 0.176828861, -0.188249394, 0.09324269, 0.094032906, -0.15741083, 0.0183089897, -0.025142502, -0.185235664, -0.105590858, 0.126755387, 0.0810155272, 0.0908192694, 0.257951409, -0.157443106, 0.205290884, -0.0489252396, -0.0989102721, 0.0708614588, 0.0386378206, 0.201516673, 0.0292547792, -0.0833374709, 0.132945493, 0.156132996, 0.00765515072, -0.190696836, 0.0847563595, -0.130459666, -0.174606368, 0.186493203, -0.185741857, 0.0914283767, -0.200763315, 0.0963705927, -0.164442599, -0.120197445, 0.0842603222, -0.187861234, 0.0992910936, -0.0723259225, 0.131771117, 0.0294709411, -0.0707816929, 0.15362066, 0.111908376, 0.078812331, 0.0535888821, 0.0507810563, 0.131110504, 0.179611921, 0.026744267, -0.0871720165, 0.0355067551, 0.118356422, -0.204518527, 0.0498766974, -0.0372236706, -0.00990310404, 0.10396497, -0.00883602072, -0.177933022, 0.0129285334, -0.12813133, 0.0643947497, -0.0221159253, -0.078253977, -0.156190872, 0.0223176498, -0.0749285966, 0.160610095, 0.0397448465, -0.144857541, 0.210528627, -0.177495837, 0.170002475, -0.0258958396, -0.113389783, 0.109926522, 0.195601434, -0.0548773855, -0.149894163, 0.148451984, 0.0346607901, 0.140283972, -0.00360311568, -0.102635242, -0.0503319688, 0.0162678473, -0.0676407441, -0.11571575, 0.112506241, -0.118930839, -0.151946649, 0.0985130519, -0.1923296, -0.0602569394, -0.037379276, -0.193716258, -0.0948935449, -0.020577101, -0.179147139, -0.195478693, 0.123371579, -0.00464495225, 0.0504263602, -0.0386064462, -0.0517891161, -0.169164538, 0.11771892, -0.0632881671, 0.125877112, 0.192654654, -0.0948174372, 0.0738299266, 0.126855522, -0.118285932, -0.0321045406, 0.0178604145, -0.0212341771, 0.148154989, 0.130340979, -0.0704322532, 0.0328871049, -0.227042913, 0.239740446, -0.0955699533, 0.114672013, -0.0708279312, 0.10800238, -0.109282725, 0.142058045, 0.105162479, -0.051887475, -0.0467856638, 0.123139441, -0.106748275, -0.175780401, -0.127217188, -0.181122348, -0.0676865727, 0.117284544, -0.0273130462, 0.0963890329, 0.00385483191, -0.177152038, -0.191867977, 0.077240102, 0.124747507, 0.0890129358, -0.0591309927, -0.121862456, -0.19205831, 0.122563228, 0.176135257, -0.177255824, 0.0381551534, 0.0424975604, -0.185359091, -0.188019961, 0.114714131, 0.161240518, -0.119956791, -0.00404445827, -0.0148509219, 0.0826404542, -0.0528445691, 0.145070598, -0.0415300168, 0.185449079, 0.0144401034, -0.0457542241, 0.121085688, 0.159310594, 0.197267592, 0.0817764252, 0.119335428, 0.0792978927, -0.137601241, -0.0160116367, -0.16096127, 0.0202337243, -0.0156570133, 0.17746596, -0.0477557518, -0.057627324, 0.165322959, -0.147759885, -0.088363573, -0.183882236, 0.216872111, -0.120255038, -0.0487861186, -0.0615872554, 0.126300633, -0.0990248471, 0.0368622988, 0.223582864, 0.0624831654, 0.010734871, -0.116444357, -0.203225613, -0.127781093, -0.166673332, 0.157802746, -0.0282158162, -0.109729975, -0.0391220339, -0.124125309, 0.0324856862, -0.175051495, -0.0247840639, 0.0936974436, -0.00736786192, 0.155662224, 0.157572389, 0.0846097469, 0.0808747634, -0.029931752, 0.130156875, -0.194955394, 0.0540007949, 0.297759801, -0.15280652, 0.0210758597, 0.0932299495, -0.167536736, 0.285581648, -0.0180603843, -0.179686129, 0.204945594, 0.189112514, 0.165582985, 0.143395647, -0.126252934, 0.0896839723, -0.298827648, 0.064478986, 0.000745264464, -0.16088663, -0.174918249, 0.0957706571, 0.0120447576, 0.119768813, 0.0807619318, 0.0893344283, -0.25136587, 0.127414092, 0.207855508, 0.0846856162, 0.0175084565, -0.10128703, 0.101297647, 0.208785698, 0.138138175, 0.0138534503, 0.0905889496, 0.13177821, 0.18886824, -0.0161923002, 0.189213589, -0.0682863444, -0.166542068, -0.00136115553, 0.0997680947, -0.0653852895, 0.146990359, 0.181544811, 0.115617692, 0.298607945, -0.0134123974, 0.145018026, -0.29561004, -0.124093696, -0.210322186, 0.137198851, 0.0914252549, -0.0175533239, 0.192823961, 0.183647707, -0.144407481, 0.0237307549, 0.175023243, 0.116533205, -0.010630399, 0.0754853338, -0.0653730035, 0.114706591, -0.159099877, -0.0851648599, -0.1207624, -0.0410666317, -0.172199935, -0.145232454, 0.16999276, -0.146817982, -0.0389965475, -0.0854866505, 0.0712565035, -0.00583642721, -0.197309196, -0.0306858718, -0.151972204, 0.0138290226, 0.201786533, -0.033470422, 0.111182824, 0.0868683606, -0.118202969, 0.0617301315, 0.132822946, -0.154013336, -0.00978311896, -0.161551476, -0.193557248, 0.0101869851, -0.126305878, 0.158561811, 0.00379236042, -0.0607737899, -0.0138211846, -0.158382684, -0.0691986978, 0.133874074, -0.201073974, -0.119042397, -0.0212140232, 0.0352598876, -0.0136535764, -0.0176571012, 0.210377857, -0.197992519, 0.0080832541, -0.00235559046, 0.095504269, -0.209513187, -0.215412378, 0.168746248, -0.215368554, -0.0952431932, -0.0601882786, -0.128752172, 0.113622233, -0.215524599, 0.201375023, -0.107492052, 0.0754652768, -0.0948438123, -0.121238068, 0.149828091, 0.161296472, -0.0535617173, 0.0448756069, 0.215061948, -0.0858141333, -0.104567416, -0.13317892, -0.180668265, 0.157652691, 0.000676110387, 0.0542567819, 0.103542104, -0.160294861, 0.0630884916, -0.0210512578, 0.0308071226, -0.108765341, 0.105836019, -0.0544864237, -0.0361126959, 0.0175312012, -0.0544892699, 0.165185824, -0.0246543884, -0.0384053588, -0.0629663616, -0.165999919, 0.0924038738, -0.0472313017, 0.178175375, 0.147123411, -0.0634953082, 0.212211952, -0.035074994, -0.0309012234, -0.0756640583, -0.0832019448, 0.14364703, 0.0768184513, 0.132498935, 0.117131457, -0.0801562518, 0.181623742, 0.19624342, -0.197934449, 0.181445286, 0.10837917, 0.126055077, 0.0945705026, -0.0554487109, -0.180778623, -0.118354313, 0.110690013, -0.15024513, -0.193064138, -0.171204776, 0.0157593787, 0.100202553, 0.214262843, -0.148953438, -0.11341837, -0.0936558172, 0.0606097542, -0.0733776987, 0.20756118, 0.0454133786, 0.211113855, 0.263197571, 0.0173376407, 0.0348490179, -0.0670863166, -0.0259215664, -0.220633924, 0.167376027, 0.30080685, 0.152899742, 0.100315377, 0.0216483381, 0.0153267374, -0.0821862444, -0.022511309, 0.110671572, -0.197649375, -0.243930042, -0.0089917779, -0.16742897, 0.25845921, 0.0806541368, -0.0169763733, -0.150612444, 0.0804499462, 0.147269264, -0.123657018, -0.101714112, 0.0392946117, 0.235302284, 0.129554257, 0.20972079, 0.00137448253, -0.160698906, 0.0453142338, 0.0750062764, -0.044447802, -0.0454354547, -0.0594326332, 0.0154880593, -0.135283649, 0.156637296, -0.0949086621, -0.204240441, 0.199247792, 0.0847830772, 0.0778177977, 0.262001753, -0.0237951018, 0.254970968, -0.103296667, 0.1293993, -0.211035922, 0.103326999, 0.000826618809, -0.0683762655, 0.156546369, -0.012880085, -0.0566472597, 0.105513714, 0.0323817059, -0.180392623, -0.0829131231, 0.275576562, -0.119350486, -0.256336868, 0.0225851666, -0.0718415678, -0.032045424, 0.157612577, 0.295247853, -0.161926433, 0.0551234297, -0.200971603, -0.149542153, -0.112447798, -0.188605458, -0.10279642, -0.185480207, 0.186702803, 0.203769177, -0.0506769307, 0.340962738, 0.0492642671, 0.00382401654, -0.295713395, 0.0791265443, 0.145609438, -0.118261933, -0.0462953039, -0.26303187, -0.167325541, 0.229171544, 0.125606567, 0.0196683183, -0.0821758062, -0.172154814, 0.134631366, 0.105954275, 0.0713844672, 0.066780068, 0.0916744471, 0.325054318, 0.134490564, -0.18094638, 0.0252105873, -0.154933974, -0.00310963392, 0.0248205513, 0.126237467, 0.014732969, -0.103780881, -0.19062826, -0.0709873661, -0.0277325865, -0.0735364705, 0.133878663, 0.0306869727, 0.197213531, 0.217959478, 0.0710183606, 0.18170689, 0.21944575, 0.0610789806, -0.116570912, 0.12491186, 0.0503248312, -0.110214539, -0.0159544032, 0.232890576, -0.0456155278, 0.00884607527, 0.187331676, 0.21877192, 0.204476058, -0.115975544, 0.0187843088, -0.09255445, -0.29152, 0.0851894468, 0.0949364305, 0.262373477, -0.0559873134, -0.0886857882, -0.107428819, 0.175252438, -0.181784943, 0.248689443, 0.0079609314, -0.155982539, -0.247614115, 0.197390601, 0.0732584447, 0.0571540222, -0.153867841, -0.185098931, -0.225856975, 0.151971042, -0.17325078, 0.166293293, 0.21347858, 0.137752622, 0.0146298427, 0.165977046, 0.200429872, 0.243356928, -0.0243835449, -0.132510141, -0.170158356, -0.210107028, 0.054322429, -0.0642425045, 0.070434615, 0.00680774171, 0.115169078, -0.0843608603, -0.113310277, -0.250803977, 0.00723329745, -0.320745975, 0.0171446204, 0.0268929899, 0.0155198043, 0.183056667, -0.0546245314, -0.0218649153, -0.107723393, -0.0206710231, -0.0810157731, -0.0866106674, 0.154913038, -0.0283856317, 0.157422259, 0.249080539, 0.197582707, 0.0180592034, -0.0630287081, 0.0954426602, -0.00257873558, 0.197637767, -0.0483088568, -0.205665752, 0.178116858, -0.215542749, 0.0139305266, -0.0284120627, 0.0472723357, 0.114193209, -0.113162771, -0.0734884441, 0.190928593, 0.14512518, -0.179998294, 0.0362271219, 0.0808228552, -0.0790003017, 0.0780607685, 0.0691427216, -0.0794865191, -0.190427512, -0.194445565, -0.117233612, -0.181705579, 0.076732479, -0.0706049204, 0.110384241, 0.109668888, 0.00635866122, -0.120385066, -0.182506919, 0.0288684703, -0.155140281, -0.00705729891, 0.0220523346, -0.0523335524, -0.127393574, -0.226881415, -0.0877430663, 0.141399264, 0.180214092, 0.0126109738, 0.104212426, -0.00757380715, 0.258023709, -0.0758938268, -0.169211, 0.0147744548, 0.0781950727, 0.0368106291, -0.278180361, -0.0971170142, 0.119301975, 0.193576843, 0.134058133, -0.0579313375, -0.0559127405, -0.0187151711, -0.0745572597, 0.0402791612, 0.11351911, 0.110996328, 0.10230045, -0.119222939, -0.0110910339, 0.0194552336, 0.14156279, 0.280852199, -0.166947231, 0.102535248, 0.0493896715, -0.0241324138, -0.176901072, -0.0267906673, 0.252696484, 0.307401866, 0.00364437792, 0.158837378, 0.263545632, 0.0133025851, -0.0667897686, -0.0859481618, 0.145068467, -0.0603770092, -0.0731502622, 0.269838184, -0.245759487, -0.0586617142, -0.0775664076, -0.208350435, 0.0898162201, 0.0956078693, -0.134778693, -0.0955108702, -0.0629637241, 0.164887547, -0.0951353088, -0.0474154986, -0.0317355469, -0.311545223, -0.034149304, -0.133716777, -0.254200995, 0.233857363, -0.221086636, -0.0875458941, 0.144417778, -0.0733914226, -0.0500378273, -0.16867502, 0.108182065, 0.128211737, -0.0357037261, 0.16355747, 0.00208666385, -0.341230929, -0.110794365, -0.192407697, -0.185402006, 0.0158167668, 0.228281468, -0.0576616935, -0.0166208204, 0.231899574, -0.0969194695, 0.176652476, 0.166342959, 0.0320710912, -0.179827735, 0.132767901, 0.0290033314, -0.152132601, -0.181854218, -0.0543435551, -0.147026494, 0.132066295, 0.000380948186, -0.046831917, -0.0122211166, 0.265439212, -0.385553628, 0.19313477, 0.133767381, 0.286021829, -0.22221379, -0.293776661, 0.148888484, -0.181432143, -0.16458258, 0.268145353, -0.204560816, 0.0846042112, -0.109482028, -0.0879192576, -0.147025988, 0.288842827, -0.088969633, -0.0655507073, 0.263407081, 0.133582711, -0.0163365304, 0.110040441, -0.0645436272, 0.0251421444, -0.10840106, 0.179400072, -0.106979035, 0.0695290193, 0.109481424, 0.210353449, -0.0532516129, -0.167095572, 0.0434949584, 0.175142482, -0.0420172065, -0.100425139, 0.165737182, -0.165261269, -0.119268917, 0.142626181, -0.188711599, 0.0471658744, -0.0998743027, 0.108773425, 0.171581998, -0.0881806239, -0.118828684, 0.0752182528, -0.185938254, 0.102960572, -0.00374448881, 0.143556684, -0.157970682, -0.0651584789, 0.126855001, 0.182917491, -0.160805538, 0.123719871, -0.0744021162, 0.213524118, -0.207614541, 0.0227269568, -0.0975663513, 0.0987157747, -0.0909273997, 0.138845056, -0.0999631882, 0.181141108, -0.180883646, 0.150684878, 0.072670795, -0.11002925, -0.120575607, -0.0391260162, -0.0647687092, 0.17848663, 0.0242926795, -0.143397227, 0.181315631, 0.115013622, -0.217152998, -0.016199477, -0.0158816669, -0.124248572, -0.12989518, -0.0339076035, 0.264628232, -0.0808567181, -0.0246815663, -0.0834978744, 0.161822602, -0.138402522, -0.00808761735, 0.0439582318, 0.154923141, 0.0127866575, 0.157803074, -0.0195006952, -0.145444661, 0.15624623, 0.213899404, -0.216991454, 0.0774733201, 0.102065235, -0.124791786, -0.207634076, -0.164074779, -0.0574968681, 0.089080818, -0.0694269165, 0.211942866, -0.114976563, 0.214145839, 0.198561743, 0.0715887323, 0.109872617, -0.0963600874, -0.079338029, 0.0805210099, 0.0106852446, 0.191253379, -0.067177996, 0.11775624, -0.110801004, -0.102861449, 0.1769429, -0.223849356, 0.0693205595, 0.145785511, -0.032342162, -0.158411354, -0.00197427161, -0.095368214, -0.188921377, -0.113391459, 0.0368723348, 0.107978091, 0.0824893937, 0.0900589675, -0.041756928, -0.064508982, -0.181163505, -0.171657398, 0.026455136, -0.199689955, 0.0629645661, -0.117474094, -0.15332523, 0.0785275772, -0.111598738, -0.103435583, -0.163627595, -0.00887487829, -0.157007217, 0.00934804231, 0.1409017, -0.000921073661, 0.0372746959, -0.174577355, -0.0164345335, 0.0782096386, -0.0826458782, 0.138327822, 0.0130521106, 0.142504245, -0.0212440453, 0.235662311, 0.292200476, -0.124307498, -0.141203091, 0.104294352, 0.265598536, -0.202951029, -0.31308794, 0.176690981, -0.316680521, 0.308380634, -0.058346685, -0.052924715, -0.068701461, 0.240178868, -0.194287747, 0.128212035, -0.121045195, 0.18089883, -0.0418058485, 0.0846816227, -0.119049914, 0.00999071915, 0.03216362, 0.127670601, -0.200703219, 0.0612659827, -0.307814896, -0.328196347, -0.119040579, -0.175974175, 0.247130468, 0.0949836671, 0.0164293498, -0.0871255696, -0.0288449004, -0.0993912593, 0.0679356381, 0.0571999848, -0.0168665498, 0.173970565, 0.00567579689, 0.206851333, -0.0155466767, 0.116136476, -0.0451772027, 0.0345146023, 0.171833515, -0.14317131, 0.0439632647, 0.0550731719, -0.174111396, 0.249948263, 0.0319778696, -0.08461494, -0.194183409, -0.0776880309, -0.0970808789, 0.0736219287, -0.13262856, -0.0557855815, 0.0211500153, -0.236246914, 0.22175169, 0.162301347, 0.0972244814, -0.176554397, 0.204008728, -0.209684461, -0.18114011, -0.1861417, 0.281658024, -0.00434876187, -0.000967082102, -0.182629734, 0.109987505, -0.0832468048, 0.0613217019, 0.148019463, 0.000290387106, -0.142763898, 0.185766563, -0.0045414567, 0.168641582, -0.156493008, -0.169194326, -0.11528603, -0.0347869396, 0.253748775, 0.0731557384, 0.037423566, 0.162255421, 0.169754088, 0.257631987, 0.165029943, 0.0698102564, 0.0314833559, 0.164437681, -0.128836766, 0.280385345, -0.132313639, 0.0832324475, -0.159102678, -0.190169424, 0.120876521, -0.0708724335, 0.108387083, -0.013849372, -0.173526362, 0.168055281, -0.0783005506, 0.133223042, -0.052906163, -0.16011405, -0.156364277, 0.170717791, -0.135527775, 0.302193105, 0.0370368697, 0.144021943, 0.152141228, 0.072664246, 0.0809864327, -0.0436896682, 0.10182593, 0.0915664807, -0.184139475, 0.280362487, -0.195510402, 0.0830965191, -0.0758729503, 0.223914117, 0.00844487827, 0.00993681513, 0.0982448608, -0.103829846, 0.00631501665, 0.0602077693, -0.229385301, 0.304050446, 0.210445672, -0.0769463331, 0.108615175, -0.0788970515, -0.127578288, 0.214681074, -0.0700043291, 0.166759819, 0.0396312959, -0.144758493, -0.106974468, -0.0965421125, 0.188366085, 0.28905794, -0.125003085, 0.248191193, -0.022866942, 0.301850051, -0.163019001, -0.328558654, -0.0491153672, 0.0805409625, -0.0996451229, 0.256436139, -0.125509635, 0.0881489664, -0.0299049839, -0.272820115, 0.0276542306, 0.072070688, 0.017024979, -0.0835376158, 0.193469211, -0.0293851048, -0.191110089, -0.0412489772, -0.208624303, -0.24148649, -0.205899239, -0.174337134, -0.0175865591, 0.298654824, -0.0985588804, 0.103253216, 0.24924536, 0.205758289, -0.196999446, -0.149646878, -0.143381536, -0.000880725158, -0.0068264748, -0.174360752, 0.249812827, 0.109578051, -0.081599012, 0.113797002, 0.079932496, -0.0615099408, 0.191720381, -0.208634764, 0.150513843, -0.0344681069, 0.218191922, 0.139449969, 0.171120629, 0.1082827, 0.163610205, 0.0875669345, -0.116561994, 0.118207827, 0.0104034245, -0.16478233, -0.0413739011, -0.316277593, -0.0421933122, 0.0120029449, -0.116558015, 0.0348773338, 0.0611173026, -0.145482197, -0.0627405196, -0.182251006, 0.0826851279, -0.0607742444, 0.0268052518, -0.0526164658, -0.0653537959, -0.179316863, 0.105216481, -0.0154515207, -0.155959472, 0.13121824, 0.25053665, 0.213652462, 0.0733022988, 0.0634803474, -0.133813843, -0.0560159571, 0.123325393, 0.169942483, -0.0188645292, -0.146081492, -0.0042090537, -0.152687699, 0.152199179, -0.0402537622, 0.150147647, -0.15232645, -0.101902142, -0.0839850903, -0.278659999, -0.146883801, -0.0142387301, -0.0918006599, 0.198642433, 0.164413884, -0.183536232, -0.0297051743, 0.159891501, -0.122745588, -0.102025181, -0.0521458909, 0.118992224, -0.060556896, 0.195035189, 0.259946346, 0.0685981214, -0.148837596, -0.0323895104, -0.0847889632, 0.182129964, 0.119295359, -0.0368872695, 0.238972053, -0.155852035, 0.167594254, -0.0925863683, 0.0172753409, 0.189614743, 0.162803963, 0.163829163, 0.215808108, 0.0124880038, 0.0426811688, -0.0600209348, 0.0615481213, 0.165346935, 0.0153156063, 0.121975742, -0.175549001, 0.183664352, 0.144022495, 0.0322715566, -0.107829265, 0.0768434852, 0.0050736377, 0.0618446544, 0.153952852, -0.169535995, 0.166753307, -0.186460227, 0.00901123788, -0.0184693541, -0.0857320651, -0.0475749783, 0.00862984639, -0.0971527323, -0.196421653, -0.0968040973, 0.238713965, -0.0107892593, 0.178670123, 0.082849972, -0.067512013, 0.103636593, -0.172591835, 0.162427366, -0.0980086103, 0.103627391, -0.00657122722, 0.196705267, -0.0885492787, -0.21484302, 0.0713789761, 0.00349842641, -0.114411183, 0.00135329366, 0.172899455, -0.0640534312, 0.176380396, 0.129859045, 0.152343497, 0.188691467, -0.0690017864, -0.137624815, 0.0596759468, 0.161572218, 0.030274827, 0.0932867527, -0.0543891117, 0.0914924815, 0.0758234411, 0.189578816, 0.216388658, 0.136622667, -0.224723607, 0.115231387, -0.143994942, -0.0134596284, 0.0285644792, -0.0765158683, -0.0898127109, -0.0216522682, -0.0452857055, -0.180066332, 0.0636309981, -0.136346862, 0.160724685, 0.104276851, -0.0502810515, 0.214406371, 0.00751658203, 0.0742831528, -0.0960830152, -0.103430808, -0.149839222, 0.122873515, -0.199809447, 0.0846741796, 0.0414155461, -0.149651155, 0.0535871387, 0.032020431, 0.00699738273, -0.12234541, -0.0605762973, 0.0471933074, -0.00849266909, 0.0234554689, -0.0544377342, 0.0270179659, 0.172541559, 0.0252916161, 0.0905541778, -0.144034952, 0.00168407825, 0.173910916, -0.0856598467, -0.0220967811, -0.0514697209, 0.0803929046, 0.127755255, 0.171276376, 0.104453139, -0.0212837942, -0.0249362309, -0.358178616, -0.233663827, 0.233707651, 0.256034017, 0.103490725, 0.00574883632, -0.0556842498, 0.131842449, 0.00785240531, 0.0435351245, -0.118263483, -0.150564089, -0.117127106, 0.015985528, 0.088842757, 0.14202477, -0.00392921269, -0.141630784, -0.108435906, 0.150415316, 0.192709893, 0.242879584, -0.187250435, 0.0510517657, 0.229519933, -0.0843288153, 0.0532751195, 0.186514959, 0.0342584439, -0.0914594829, -0.0284124669, 0.141796708, 0.00305303931, -0.0396114551, -0.115827665, -0.12504971, 0.231261835, 0.135242477, -0.0376397893, -0.146970883, 0.233937755, -0.114139147, 0.156069487, 0.179028809, 0.178957433, -0.0414629728, -0.0976045877, 0.0569484569, 0.103674464, -0.089665994, 0.0826087892, -0.105914153, -0.00952274725, 0.185328886, -0.0473689064, 0.171411321, -0.135359928, 0.237343296, -0.293576032, 0.0484540462, 0.0989309847, -0.12313319, 0.21306318, 0.0288836546, 0.0259658769, -0.0176200364, 0.202105507, 0.239969552, 0.125312254, 0.0684467033, -0.189783171, 0.024794735, 0.107969731, 0.17213501, -0.0679843202, -0.176238269, 0.00562783564, 0.198162049, -0.0273213014, -0.229449779, -0.0726197436, -0.146376207, 0.0733661801, -0.122138776, 0.0300521944, 0.000627006986, -0.224758834, -0.219826937, 0.042535685, -0.11363896, 0.0945541859, 0.118705377, 0.0555131733, -0.329797447, 0.0684644952, 0.260578483, -0.0437527634, 0.0811403245, 0.0408508256, 0.15580976, -0.0451794863, 0.0944328681, 0.199969038, 0.0696579441, 0.223595411, -0.0154632749, 0.321737945, 0.251616448, -0.0567427538, 0.035431765, 0.280902177, -0.169113502, -0.231067359, 0.0143873319, 0.0581891723, 0.154215962, 0.0250351746, 0.238159895, 0.128872484, -0.221735775, -0.0697579384, -0.075381659, -0.0484818742, -0.0863361508, 0.123765059, -0.135387972, 0.231054485, -0.0443002544, -0.243541643, 0.151080266, -0.106428668, 0.0855598897, 0.0846331418, -0.0779921785, 0.0547915027, -0.0920602605, 0.0887217745, -0.0030759566, 0.0840683505, -0.0667907745, 0.0150866825, -0.113728702, 0.0240516253, 0.0788644105, 0.0189627409, 0.029980829, 0.182710513, 0.233252287, -0.0950233042, 0.0486974977, 0.0204964131, -0.0657696128, 0.242969364, 0.034332294, -0.123168163, 0.246184021, 0.0397303998, 0.028434189, -0.115440212, 0.0868595541, -0.145101041, 0.0786464363, 0.0524663962, 0.0946072713, -0.160390154, 0.268412858, -0.202053457, 0.170204252, -0.141202495, -0.209169641, -0.0217667911, -0.276255965, -0.208408445, 0.0612591468, 0.18525213, -0.0280163027, 0.0532558374, 0.038261883, -0.111344911, 0.0510275178, 0.137613237, -0.0182486102, 0.022279419, 0.237698808, -0.168505922, -0.0947840884, -0.0860128328, 0.0939792022, 0.0062875296, 0.290792286, -0.178391397, 0.0912785605, -0.071976088, 0.180548236, -0.196116716, -0.154281169, -0.0599976256, 0.261835635, 0.0432700068, 0.244295612, -0.222427472, 0.0652513355, -0.17671591, -0.203425258, -0.131267071, 0.0277503077, -0.261542737, -0.002615412, 0.295612812, 0.0422270782, 0.169738501, -0.136077911, -0.241452679, -0.158954144, 0.0203940291, -0.0218450259, -0.21398285, 0.260178745, 0.0980303138, 0.00973836519, -0.257299483, 0.224123374, 0.0211241115, 0.18352662, -0.064140141, 0.0862681791, -0.163428918, -0.152894586, -0.00333995232, 0.0032048868, -0.0328324623, 0.0929068178, -0.279507995, -0.0916615948, 0.149792582, 0.0819854364, -0.0381851047, -0.0611945577, -0.134679809, 0.0265907645, -0.106183901, -0.0546292849, 0.212225929, 0.155997798, 0.0469628684, 0.0114867613, 0.0375453793, -0.0232304651, 0.201258332, 0.0445280969, -0.108712807, 0.0448913462, -0.0595548563, -0.00239899638, 0.055149626, -0.00122337963, -0.0738636926, -0.081668295, 0.202223718, 0.136749536, -0.227384835, 0.0613598339, -0.115820222, 0.0364864096, 0.0139585184, -0.0280776732, 0.180970713, -0.046631746, 0.0747796074, 0.126691923, -0.0111388853, 0.107929185, -0.0551268123, -0.0529108122, -0.212241918, 0.136584833, 0.155696839, 0.0378725938, -0.151348546, 0.00820482895, 0.0856666714, 0.137337208, 0.147699654, -0.0763601139, -0.0242069904, -0.0654426292, 0.0947293192, 0.0777328461, 0.0894588232, -0.124189667, -0.197469324, 0.18639116, 0.0779219195, 0.141812861, -0.0726427585, -0.194079414, 0.0403500609, 0.0486738719, 0.175959468, -0.0224688575, 0.108159691, 0.110468484, 0.0989225358, -0.0435029604, 0.0932252854, 0.0202672239, -0.0806071311, -0.0692079961, 0.21573095, 0.165748715, 0.0341887586, 0.196531609, -0.106021568, 0.0170011446, 0.0364869945, -0.0480184555, 0.160415426, 0.238614678, 0.0291153304, -0.0692989081, -0.329096109, -0.0360180438, 0.256817967, 0.225853592, -0.224268287, 0.175842762, -0.198225558, 0.0573723502, -0.0511965454, 0.117915072, -0.0368777364, 0.0182616115, -0.00727006095, -0.0168267079, -0.0614160858, 0.156759843, 0.162976161, -0.00199627364, -0.17093797, 0.201199114, -0.194492713, 0.0589784794, 0.0552661046, -0.167786106, 0.140908763, -0.068700999, 0.0502691977, 0.0795648023, 0.0274966806, -0.296720952, -0.163464576, -0.102106683, -0.00985952932, 0.109491237, 0.00823518075, -0.197602898, 0.241903737, 0.0013750908, -0.168662667, -0.123866923, -0.204145133, 0.0930801407, 0.328670114, 0.00163828232, 0.220920488, 0.0642628074, 0.328812987, -0.0748362392, -0.0226152278, 0.000289303658, 0.188728347, -0.0364874303, -0.0651446581, 0.231653139, 0.0857582167, -0.194839388, 0.0351886451, -0.0548176616, 0.0118231382, -0.148435593, 0.0464327261, -0.0904112831, 0.0666049942, -0.209124938, 0.0648437589, 0.182237193, 0.214572534, -0.00191250537, -0.1671011, -0.110546388, -0.154530227, -0.106844932, -0.0305259917, 0.116241798, 0.109203883, 0.142477855, -0.0726438016, 0.0829489529, 0.0612219125, 0.0201825909, -0.131854653, -0.225124791, -0.129626438, -0.0346009545, 0.205493644, -0.123570427, -0.0745602846, -0.187618464, 0.13536644, 0.176973596, 0.234079748, 0.0889393911, -0.0863182768, 0.165225297, 0.137968197, 0.279592723, 0.0361696146, -0.173749968, 0.0601600967, 0.0129619762, 0.208610386, 0.220640108, -0.115378678, 0.0240061432, 0.278004318, -0.0265378393, 0.149464399, -0.303708673, -0.105789356, 0.0307838731, 0.193645462, -0.165561646, -0.0895986408, -0.0594347157, 0.254087687, -0.0558889918, -0.106389455, -0.00137458323, -0.194988936, 0.0805720314, -0.0352395177, 0.194134623, -0.116110273, -0.174519628, 0.0278469343, 0.0595925637, -0.130331695, -0.0923151374, 0.0643297732, -0.177647516, 0.10481973, 0.192607358, -0.141913235, 0.0599878654, -0.154343843, 0.264552563, -0.0673295557, 0.183654264, 0.179233626, 0.00202305615, -0.33549431, -0.156067759, 0.116495214, 0.164007157, -0.0761157051, 0.0759984627, -0.137309909, -0.0688316524, 0.154320285, 0.249968484, -0.219860017, -0.325449139, -0.129957005, -0.326592982, 0.205126315, 0.0471690372, -0.113722183, 0.101460293, -0.132077157, 0.0266415607, 0.00812615175, -0.179480046, 0.162329659, -0.0515648499, 0.315276504, -0.00411519269, -0.02481113, -0.0660336092, 0.20307903, 0.116764992, 0.145217434, 0.231170014, 0.129283935, 0.227875918, 0.335049301, 0.169715032, -0.0661990941, -0.222038403, 0.112036951, 0.118910842, -0.214670569, 0.0934555307, 0.0968824625, -0.150049731, 0.149248824, -0.0754649118, 0.273794323, 0.0952707529, -0.29306978, -0.157772511, 0.135602057, 0.14062117, 0.369418502, -0.0413367189, 0.0816308931, -0.278485179, -0.0156329628, -0.353450298, -0.0292544812, -0.262566298, 0.0992213935, -0.170477495, 0.127993777, 0.165333867, 0.197797731, 0.250114858, 0.104357131, 0.0609139763, -0.390009731, 0.095229812, -0.106860213, -0.1796031, 0.13155356, 0.00892605539, -0.189845622, 0.179488435, -0.129862547, 0.0306370258, 0.000393755792, 0.183470011, 0.201606512, 0.00992667116, 0.138476804, -0.0199141521, -0.0361978561, -0.00738017075, -0.173073292, -0.136918575, -0.221550018, 0.16833882, 0.0337039381, 0.193500176, 0.121161528, -0.0153150447, -0.229320586, -0.162542269, -0.103140332, -0.0991333276, -0.21625343, -0.122940831, -0.0816918612, 0.292686313, -0.126720279, -0.245018229, 0.156526193, 0.231272772, -0.12768504, 0.046446193, -0.135035276, 0.237224385, -0.207771942, -0.165304184, 0.0449262112, -0.16046451, 0.0515512154, 0.0247535985, 0.179941446, 0.141006634, 0.148099631, 0.0461900011, -0.125380158, -0.260761499, -0.0365008488, -0.175376043, 0.173839927, 0.0840524882, 0.150757536, -0.00193478167, 0.134457171, 0.0838706568, 0.19708553, -0.108223915, -0.214755952, -0.180884525, -0.210335225, 0.198198155, -0.0710237324, -0.18349649, -0.10621804, -0.0015054564, -0.0930908322, -0.0695800856, 0.120227791, -0.0628320128, 0.161675051, -0.0369836837, -0.104480736, -0.115745157, 0.113166645, -0.226809382, 0.0440124832, -0.0557170361, -0.00395971676, 0.15534845, 0.116499223, 0.190032437, -0.105497465, -0.26288572, 0.0491223671, -0.219523475, 0.164801389, 0.0884424895, -0.180786639, -0.0025313925, 0.107427284, -0.015959831, 0.280966669, -0.101899825, 0.0844253153, 0.214183345, -0.0680119321, 0.0215379167, -0.215002313, 0.103997082, 0.0602454916, 0.162121207, 0.223211929, 0.0564612225, -0.0155185293, -0.0849888176, 0.0710228682, -0.0188842621, -0.0679497048, 0.228468344, -0.168624103, -0.187010109, -0.0338806175, 0.0473464616, 0.156233341, 0.210370451, -0.162648752, 0.0154813081, 0.0151715912, -0.224204272, 0.162158608, -0.212012723, 0.108205117, 0.120467298, 0.0116960257, 0.0391680412, -0.120638661, -0.0434363931, -0.0632359162, -0.18498835, -0.0534989648, -0.104398511, 0.14394021, -0.0630829409, -0.202434331, -0.221765876, 0.170155361, 0.146729127, 0.136266768, 0.0854845718, 0.00931845978, -0.0396513678, 0.243059888, -0.0143531486, -0.213143229, 0.163626105, 0.228435755, 0.0763803273, 0.294812024, 0.0303754285, 0.0224024169, 0.103866428, -0.0755221769, -0.146329269, 0.187158212, -0.0402141139, 0.215759218, 0.0578194857, 0.00068547955, -0.189536303, -0.157405496, -0.0117263664, -0.171880484, -0.0894706845, -0.195492998, -0.115787826, 0.106829114, -0.0732092932, -0.106249996, 0.0644781068, 0.0493799672, 0.0191225074, 0.199877992, -0.154181615, -0.169715717, -0.202959687, 0.0045042932, -0.139033392, -0.107659563, -0.174030259, -0.0516406633, -0.166010961, 0.136116982, -0.0560865402, -0.116511792, -0.0237821639, -0.0764931142, 0.0603490248, -0.154312968, -0.0190427899, -0.0848358423, -0.120311961, -0.0347254574, 0.0647674352, -0.113835506, -0.177448601, -0.0797593594, 0.234833598, -0.132981062, -0.132999331, -0.0635919347, 0.030990012, 0.17009069, 0.201166883, 0.187781587, -0.203566208, -0.163287312, 0.0935856551, -0.0598677248, 0.152191803, 0.114821628, -0.0730218515, 0.231914148, 0.0966452584, 0.166506305, -0.130623624, -0.0707645714, -0.129302263, 0.119527809, 0.0635081604, -0.112864114, 0.22138299, -0.0632478669, 0.114700712, -0.0792448521, -0.0765444115, -0.119066864, 0.0346016809, 0.303022891, -0.0871448815, -0.158137739, -0.228525937, -0.208690599, 0.171160266, 0.228543878, 0.198012307, 0.0903932974, 0.0979876369, 0.0818847567, -0.337730318, -0.202390894, -0.186501443, 0.1508746, -0.231906936, -0.0942646489, 0.0780744776, 0.00662959693, 0.368186593, 0.0524481647, 0.218401685, -0.0444435291, -0.0281022284, 0.117386088, -0.139238194, 0.344955772, -0.210472822, -0.185517386, 0.0432206802, 0.067795001, 0.18226862, -0.100125775, -0.108723685, 0.313094884, 0.102345057, -0.189623743, 0.119116165, 0.117150754, 0.113522097, -0.0974836648, 0.196477339, -0.299250156, -0.206788749, 0.127461419, -0.136677414, -0.00462659309, -0.082354337, 0.118807323, -0.267264903, -0.107201517, -0.257277042, -0.0105558699, 0.177996054, -0.0946902111, 0.00526810158, -0.0918765366, 0.180687875, -0.256947458, 0.0339876749, -0.0132435262, 0.0372189954, 0.0656750351, 0.123526566, -0.124181502, -0.127795756, 0.133546874, 0.267100155, -0.138555005, 0.112637945, 0.217483208, 0.250305533, -0.221768856, 0.0510481521, -0.0648338422, -0.135197312, 0.163345799, -0.0996528119, -0.295478195, 0.221370354, 0.0090700984, 0.163102254, 0.257673502, 0.0321548171, -0.218750283, -0.0417411365, 0.141176626, 0.0455146618, -0.139999777, -0.210085616, -0.0207382087, 0.159851059, -0.0191368647, 0.0799145848, -0.191577971, 0.222179979, 0.145579785, -0.124980874, 0.00011860668, -0.0531942584, -0.101949774, -0.149084419, 0.150167912, 0.242624894, 0.158585533, 0.0457630903, 0.121281974, 0.12134584, 0.174273595, 0.0234531015, 0.0101215569, 0.261128306, 0.130410358, -0.0646373257, 0.0671577677, 0.204333737, -0.171613261, -0.147265777, -0.0430774093, -0.206877887, 0.0973792225, 0.188770488, 0.0926625952, -0.369100392, -0.169856474, 0.0436665379, 0.0837029666, 0.07298664, 0.0201208107, -0.00663427031, -0.193593293, -0.0612708442, -0.269489616, 0.247763708, -0.0919435471, 0.122422889, 0.0842806175, 0.143494427, -0.040064469, -0.0293035377, 0.205288514, 0.138122469, -0.0655390397, 0.0721975565, 0.0538080819, -0.21350269, 0.121420853, 0.167736843, -0.183765441, 0.140039474, 0.234994337, 0.118522629, -0.0847690701, -0.155740887, -0.0549678095, 0.176273555, 0.12771441, 0.20569995, -0.189131141, 0.246775582, -0.040186435, -0.322248131, 0.00692595076, 0.251584858, -0.213374496, -0.195615217, 0.110311486, 0.259365857, 0.163353637, 0.123199798, -0.0378120169, -0.132168457, -0.146660343, -0.0177994464, -0.246754944, 0.347066194, 0.19430016, -0.0613136515, -0.105118059, 0.0349555612, -0.058653295, -0.0533792377, 0.0502194315, -0.0630996078, 0.0870997682, 0.193092287, -0.131634429, -0.228073478, 0.104649357, -0.0285898186, 0.0438296646, -0.142033562, 0.291676372, 0.0511058569, -0.010557062, -0.192678869, -0.0147832278, 0.333403051, -0.0420459956, -0.100109242, 0.134338498, -0.302299052, 0.0362847596, -0.301566482, -0.108434819, -0.207868457, 0.00391505705, 0.0137217129, -0.121070772, 0.151565805, -0.044486735, 0.304707795, -0.14781113, 0.0983222872, -0.238438904, 0.181199268, 0.0213714615, 0.00745414849, -0.0138446372, 0.086607568, -0.2248061, 0.0525689647, -0.022581771, 0.127698556, -0.00474502984, -0.0635372624, 0.296566814, 0.210853308, 0.133739591, 0.130687475, 0.03697237, 0.292883813, 0.157273754, -0.208699256, 0.103416078, 0.0554397516, -0.113555133, 0.0835159272, -0.1598773, 0.274341464, -0.153718844, -0.307261914, -0.314996988, -0.107934706, -0.287681222, -0.035695672, 0.0989629477, -0.0371217392, 0.142067209, 0.117525682, -0.185213074, 0.203321055, 0.103918776, 0.0360467881, 0.120570228, 0.0285809934, 0.0886411518, -0.0242966563, -0.202274486, -0.201233998, 0.0909243077, 0.000505506992, 0.195792988, -0.0434714705, 0.113136664, -0.0384105146, 0.0505792052, 0.147569552, 0.190747276, 0.0668908209, 0.0549472421, -0.111488663, -0.211737052, 0.180603728, -0.131985426, 0.1968918, -0.140003681, -0.159247667, -0.00467215478, -0.0768030286, 0.0416528136, 0.00666475296, -0.0831374228, 0.155933574, 0.0554835647, 0.0206790417, -0.151442379, -0.115788847, 0.0548514277, 0.0478165597, 0.0842054039, 0.129231438, -0.127966464, 0.147413924, 0.160519347, -0.00875259936, 0.0528210849, -0.0149530768, -0.010312736, 0.0383928567, -0.0103502572, 0.173571721, -0.0675502419, -0.0821278989, 0.116765901, 0.184800014, 0.17291145, -0.153413668, -0.0583886206, -0.122146413, 0.0483285636, 0.214191243, -0.205721736, 0.0823977888, 0.186194047, 0.118455581, -0.149338216, 0.0548166111, -0.0753933787, 0.0112254014, -0.0632569268, -0.144131511, 0.0945755616, 0.0224814937, 0.148579076, -0.0765286684, -0.0323213264, 0.0190389734, -0.107433006, -0.0821404457, -0.154118061, -0.210388929, 0.183495998, 0.0224975739, -0.0916404799, 0.0510140248, -0.0535344146, -0.192821115, -0.0450939275, 0.0833480209, 0.0689259619, 0.0424399003, -0.195493177, -0.108997151, -0.0964532495, -0.0500763245, -0.147860095, 0.0783045068, -0.0543835349, 0.00557268132, -0.0267649665, -0.179763988, -0.0538775064, 0.204667524, 0.0844915882, -0.0702664182, -0.128816217, 0.211553112, -0.20460856, -0.147548541, -0.198193178, 0.192208156, 0.0597049594, -0.144142136, -0.0617672056, -0.0503715128, -0.110759683, 0.0165932272, 0.0270641912, 0.0965968892, 0.150237605, -0.114341743, 0.0793848187, 0.156279072, -0.0775704384, -0.190129012, -0.154963881, 0.216353029, -0.126338452, 0.0519051328, -0.113659844, -0.199669346, 0.0344904214, -0.191059664, 0.102345951, -0.148214802, 0.0581426844, 0.00217875326, -0.0605221391, -0.00890331902, 0.166813642, 0.0926778764, -0.0694191083, -0.0983804986, 0.12547265, -0.14267537, 0.180269465, -0.143098682, -0.13022919, 0.0738431364, -0.163979337, -0.17442669, -0.0242187474, -0.114045739, 0.0767761916, -0.10504967, 0.0503751151, 0.0866678208, 0.00773401279, 0.00430884957, -0.120525025, -0.176838011, -0.0863500014, 0.00866668671, -0.168607041, -0.121515945, 0.14867647, 0.185887799, 0.15785116, 0.140664503, -0.0884601921, 0.0231291223, 0.0829577744, 0.0892267004, -0.197772995, 0.189196065, -0.118800618, 0.0732194334, 0.207739875, -0.103173129, -0.065648064, -0.128727034, -0.110486537, 0.054653123, 0.0793437958, 0.15447484, 0.148488969, 0.120917305, 0.0801374763, -0.129399568, -0.156592786, 0.0600291751, -0.156443983, 0.145239115, -0.0512111932, -0.0894358903, -0.204157606, -0.168812051, -0.108613163, -0.0171637479, -0.105808534, 0.123665437, 0.0821540356, 0.0144526726, -0.142738879, 0.0227865372, 0.0507515483, -0.105444357, 0.155019537, -0.207505211, 0.0971339568, -0.0339849778, -0.0463138744, -0.0321208723, 0.132046655, 0.0198223144, 0.106232792, 0.191176817, 0.00686157215, 0.067138955, -0.145373166, 0.163319066, 0.0499063581, -0.0990407094, -0.197167978, -0.0268944018, 0.145822719, -0.083871156, -0.209732011, 0.157422855, -0.00245159306, -0.0771522969, 0.199315846, -0.149281859, 0.049090676, 0.191661701, 0.158315614, -0.0693620294, -0.0132011902, 0.125350296, -0.0149667272, 0.160916612, 0.11119552, 0.157676488, 0.0098877456, 0.189075068, 0.168989629, -0.173922271, 0.121548429, -0.195168272, 0.202848047, 0.165604517, 0.156058118, 0.0950093716, -0.127327457, -0.111984469, -0.0613512285, 0.0418962389, -0.197636545, -0.114189513, 0.126012728, 0.155268207, 0.0866028816, -0.0889877826, 0.112122208, 0.194389224, 0.112043038, -0.069294557, 0.0346671753, -0.176826715, -0.203006268, -0.150415093, -0.0750610828, -0.0581135936, 0.163826838, -0.029669594, 0.109058082, -0.0119882217, 0.142015621, -0.0904931426, -0.0186770707, -0.0259640589, 0.0281509385, 0.0239989404, 0.116667978, 0.102750033, 0.091286853, -0.0383565463, -0.163616955, 0.187580332, 0.0162753612, -0.0314784348, 0.117369078, 0.0864375383, 0.100502871, -0.148412943, 0.0571034662, -0.0606366396, -0.161042437, -0.0797111019, -0.0348239429, 0.0452777334, 0.0193986744, 0.180022672, -0.00376706664, -0.075681217, 0.213514671, -0.00990024209, 0.188225329, -0.160626784, 0.0900792852, 0.18271482, -0.00601695525, 0.0461863279, -0.120181017, -0.107822776, 0.180234715, 0.100609951, -0.0603300333, -0.159216747, -0.102589242, 0.154994428, -0.0520614609, -0.183861494, -0.0509034172, -0.12675713, -0.0341059603, -0.0555140488, -0.0641053393, 0.0598824546, 0.0111815166, 0.00291509368, 0.17496188, 0.108429745, 0.115839042, 0.134348467, -0.00350385834, -0.282030761, -0.0406435393, 0.0446432419, -0.0427427255, 0.0944782719, -0.0354864225, -0.0111428648, -0.102770053, 0.0271255691, 0.242358834, 0.0536113046, 0.0741038397, -0.2916601, 0.0509373099, 0.0901637748, 0.102783382, -0.287690729, -0.0950423926, 0.0449632443, 0.0110642808, 0.140485168, 0.155553728, 0.257394135, 0.200602695, -0.0335011818, 0.105191864, -0.0773999244, 0.109473541, 0.117318951, 0.0171118602, -0.0794980526, -0.0106161162, -0.0825806633, 0.210200682, 0.049644243, 0.124389246, -0.134129956, 0.107796527, -0.214387313, -0.0956629068, 0.0328465402, -0.0811204761, -0.028460307, -0.128131568, -0.0982517526, -0.0257387385, -0.106076196, 0.0542545803, -0.151404768, 0.124424778, 0.0499416552, -0.177569553, 0.130988628, -0.304376811, -0.19533141, 0.218535423, 0.0927173048, -0.0933397934, -0.0590848438, -0.12533696, -0.182256982, 0.0507504232, 0.350399882, -0.105347395, 0.0997362882, 0.183351919, 0.223954976, 0.0116671519, 0.0770847723, 0.00941148866, -0.0585605204, -0.0564582013, -0.104068607, 0.267437309, 0.0964651331, -0.182642788, -0.189770326, -0.215519488, 0.157907411, -0.131437048, -0.10699293, -0.188718796, 0.0486624055, 0.127689123, -0.248873338, 0.078462258, -0.144253984, 0.129576817, -0.301556379, -0.114970237, 0.173650026, 0.112776645, 0.11526338, 0.115009017, -0.00548774051, 0.154869318, -0.0198779032, -0.162775025, -0.199682802, 0.135350138, 0.00967035349, 0.299527019, 0.218109444, 0.0262131374, -0.115798198, 0.272563934, -0.194497794, 0.143630132, 0.117160715, -0.214732021, 0.268078536, -0.262342006, -0.0561750121, 0.0062987851, 0.0484048985, -0.175266072, -0.0120564355, 0.243626311, -0.0441008434, 0.0145799173, 0.233922571, 0.00730382605, -0.156657904, 0.172205657, 0.221002415, 0.0211234111, -0.0905548707, 0.10886354, 0.118684202, 0.180481613, -0.0196608324, -0.178598583, 0.142019391, -0.0121234935, -0.146662265, 0.0912220255, 0.181317791, -0.16972439, 0.309380949, 0.153544962, 0.038100563, 0.192058325, -0.0871640146, 0.0492480472, 0.0830729306, -0.0759055465, 0.103810854, -0.255007654, 0.197088823, -0.0743090287, -0.21577549, -0.20244053, 0.210097998, 0.0616604239, -0.111432828, 0.184095949, -0.116312213, -0.0247057155, 0.0876967981, 0.109860271, -0.0928253531, -0.133457661, -0.177713558, -0.299925268, -0.0404093228, -0.162057132, -0.108176261, 0.12602371, 0.168155134, -0.0107569452, -0.110608943, 0.0278297774, 0.140921056, 0.112561956, 0.175497711, 0.183747575, -0.212413877, -0.130428985, 0.165591776, -0.0292511694, -0.141024932, -0.0634911358, 0.0630419105, 0.00752701424, -0.0684755668, 0.181002468, -0.102659136, 0.22071445, 0.0109583735, -0.062734507, 0.181735635, 0.184093043, 0.0399840549, 0.036717698, -0.205652788, -0.0349973813, -0.0381838493, -0.201135337, 0.138336897, 0.222890869, 0.204514265, -0.00664423173, 0.196919546, -0.0901932046, 0.0649525076, 0.00495409453, -0.0845536739, 0.0522219203, 0.0688513219, 0.129477873, -0.0250788908, -0.186325192, -0.0678296313, 0.0842106491, 0.105310403, -0.00730011286, 0.223297685, -0.128638223, -0.0857560188, 0.190256432, 0.181896374, 0.164745301, -0.208486781, 0.253901631, 0.205723599, -0.110545166, 0.177340835, 0.0701723173, -0.141629741, 0.0132791987, -0.0979559645, -0.203919381, -0.147979751, -0.0696999133, 0.0551467761, -0.148070619, 0.131242305];
